	//Alarme Rosca de PO 1
	AL_RPO1 AT %QX3200.0:BOOL; 
	//Alarme Rosca de PO 2
	AL_RPO2 AT %QX3200.1:BOOL; 
	//Alarme Rosca de PO 3
	AL_RPO3 AT %QX3200.2:BOOL; 
	//Alarme Rosca de PO 4
	AL_RPO4 AT %QX3200.3:BOOL; 
	//Alarme Rosca de PO 5
	AL_RPO5 AT %QX3220.4:BOOL;
	//Alarme Rosca 6 Horizontal
	AL_RC6H AT %QX3200.5:BOOL; 
	//Alarme Rosca 7 Inclidada
	AL_RC7I AT %QX3200.6:BOOL;
	//Alarme Balança de solidos 1 descarga
	AL_BLS1D AT %QX3200.7:BOOL; 
	//Alarme Balança de solidos 2 descarga
	AL_BLS2D AT %QX3201.0:BOOL; 
	//Alarme Balança de solidos 3 descarga
	AL_BLS3D AT %QX3201.1:BOOL; 
	//Alarme Balança de solidos 4 descarga
	AL_BLS4D AT %QX3201.2:BOOL; 
	//Alarme Balança de solidos 5 descarga
	AL_BLS5D AT %QX3201.3:BOOL; 
	//Alarme Balança de liquidos 1 descarga
	AL_BL1D AT %QX3201.4:BOOL; 
	//Alarme Balança de liquidos 2 descarga
	AL_BL2D AT %QX3201.5:BOOL; 
	//Alarme Balança de liquidos 3 descarga
	AL_BL3D AT %QX3201.6:BOOL; 
	//Alarme Balança de liquidos 4 descarga
	AL_BL4D AT %QX3201.7:BOOL; 
	//Alarme Balança de liquidos 1 rapida
	AL_BLL1R AT %QX3202.0:BOOL; 
	//Alarme Balança de liquidos 1 lenta
	AL_BLL1L AT %QX3202.1:BOOL; 
	//Alarme Balança de liquidos 2 rapida ]
	AL_BLL2R AT %QX3202.2:BOOL;
	//Alarme Balança de liquidos 2 lenta
	AL_BLL2L AT %QX3202.3:BOOL;
	//Alarme Balança de liquidos 3 rapida
	AL_BLL3R AT %QX3202.4:BOOL; 
	//Alarme Balança de liquidos 3 lenta
	AL_BLL3L AT %QX3202.5:BOOL; 
	//Alarme Balança de liquidos 4 rapida
	AL_BLL4R AT %QX3202.6:BOOL; 
	//Alarme Balança de liquidos 4 lenta
	AL_BLL4L AT %QX3202.7:BOOL; 
	//Alarme Mexedor principal
	AL_CFMXP AT %QX3203.0:BOOL; 
	//Alarme Mexedor espera
	AL_MXE AT %QX3203.1:BOOL; 
	//Alarme Bomba oleo combuALivel
	AL_BOCOMB AT %QX3203.2:BOOL; 
	//Alarme Bomba diesel para piloto
	AL_BDP AT %QX3203.3:BOOL; 
	//Alarme Bomba de baixa ligada
	AL_BB AT %QX3203.4:BOOL;
	//Alarme Bomba de alta 1
	AL_BA1 AT %QX3203.5:BOOL; 
	//Alarme Bomba de alta 2
	AL_BA2 AT %QX3203.6:BOOL; 
	//Alarme Bomba de alta 3
	AL_BA3 AT %QX3203.7:BOOL; 
	//Alarme Moinho - Estrela
	AL_MHE AT %QX3204.0:BOOL; 
	//Alarme Exaustor estrela FM1
	AL_EXFM1_E AT %QX3204.1:BOOL; 
	//Alarme Exaustor FM2
	AL_EXFM2 AT %QX3204.2:BOOL; 
	//Alarme Exaustor FM3
	AL_EXFM3 AT %QX3204.3:BOOL; 
	//Alarme Esteira TC3 Dry Mix
	AL_TC3 AT %QX3204.4:BOOL; 
	//Alarme Esteira saida Air Lifit
	AL_ESTSAIRLF AT %QX3204.5:BOOL; 
	//Alarme Air Lifit
	AL_AIRLF AT %QX3204.6:BOOL;
	//Alarme Elevador 2
	AL_EL2 AT %QX3204.7:BOOL; 
	//Alarme Esteira TC8
	AL_ESTTC8 AT %QX3205.0:BOOL;
	//Alarme falta de pressão bomba de alta 1
	AL_FPBA1 AT %QX3205.1:BOOL;
	//Alarme falta de pressão bomba de alta 2
	AL_FPBA2 AT %QX3205.2:BOOL;
	//Alarme Moinho - Triangulo
	AL_MHT AT %QX3205.3:BOOL; 
	//Alarme valvula retorno não abriu
	AL_VLRNA AT %QX3205.4:BOOL;
	//Alarme valvula retorno não fechou
	AL_VLRNF AT %QX3205.5:BOOL;
	//Alarme bomba de transferencia
	AL_BBTRANS AT %QX3205.6:BOOL;
	//Alarme Exaustor triangulo FM1
	AL_EXFM1_T AT %QX3205.7:BOOL; 
	//Alarme bomba Blend	
	AL_BBLEND AT %QX3206.0:BOOL;
	//Alarme bomba Silicato
	AL_SILI AT %QX3206.1:BOOL;
	//Alarme exaustor da torre
	AL_EXTORRE AT %QX3206.2:BOOL;	
	//Alarme geral
	AL_GERAL AT %QX3206.3:BOOL;	
	//Alarme ventilador queimador
	AL_VENTQUEIMADOR AT %QX3206.4:BOOL;
	//Alarme falta oleo bomba alimentacao
	AL_BOCOMBFALT AT %QX3206.5:BOOL;
	//Alarme Exaustor estrela FM2
	AL_EXFM2_E AT %QX3206.6:BOOL; 		
	//Alarme Exaustor triangulo FM2
	AL_EXFM2_T AT %QX3206.7:BOOL;
	//Alarme Ventilador estrela FM2
	AL_VEXFM2_E AT %QX3207.0:BOOL; 		
	//Alarme Ventilador triangulo FM2
	AL_VEXFM2_T AT %QX3207.1:BOOL;
	//Alarme Peneira 1 não ligou
	AL_PN1 AT %QX3207.2:BOOL;	
	//Alarme Peneira 2 não ligou
	AL_PN2 AT %QX3207.3:BOOL;
	//Alarme Peneira 3 não ligou
	AL_PN3 AT %QX3207.4:BOOL;
	//Alarme Peneira 4 não ligou
	AL_PN4 AT %QX3207.5:BOOL;	
	//Alarme esteira saida torre não ligou
	AL_ESTSAITORRE AT %QX3207.6:BOOL;	
	//Alarme tempo de descarga balança de solido 1 ultrapassado
	AL_DESCARGA_BLS1 AT %QX3207.7:BOOL;		
	//Alarme tempo de descarga balança de solido 2 ultrapassado
	AL_DESCARGA_BLS2 AT %QX3208.0:BOOL;		
	//Alarme tempo de descarga balança de solido 3 ultrapassado
	AL_DESCARGA_BLS3 AT %QX3208.1:BOOL;		
	//Alarme tempo de descarga balança de solido 4 ultrapassado
	AL_DESCARGA_BLS4 AT %QX3208.2:BOOL;
	//Alarme tempo de descarga balança de solido 5 ultrapassado		
	AL_DESCARGA_BLS5 AT %QX3208.3:BOOL;
	//Alarme tempo de descarga balança de liquidos 1 ultrapassado		
	AL_DESCARGA_BLL1 AT %QX3208.4:BOOL;	
	//Alarme tempo de descarga balança de liquidos 2 ultrapassado	
	AL_DESCARGA_BLL2 AT %QX3208.5:BOOL;		
	//Alarme tempo de descarga balança de liquidos 3 ultrapassado
	AL_DESCARGA_BLL3 AT %QX3208.6:BOOL;		
	//Alarme tempo de descarga balança de liquidos 4 ultrapassado
	AL_DESCARGA_BLL4 AT %QX3208.7:BOOL;	
	//Alarme no sistema do queimador
	AL_QUEIMADOR AT %QX3209.0:BOOL;
	//Alarme Bomba de Sulfonico		
	AL_BBSULFONICO AT %QX3209.1:BOOL;
	//Alarme Bomba de Agua		
	AL_BBAGUA AT %QX3209.2:BOOL;
	//Alarme Bomba de Soda		
	AL_BBSODA AT %QX3209.3:BOOL;	
	//Alarme Peso alto BLS1
	AL_PESO_ALTO_BLS1 AT %QX3209.4:BOOL;		
	//Alarme Peso alto BLS2
	AL_PESO_ALTO_BLS2 AT %QX3209.5:BOOL;
	//Alarme Peso alto BLS3
	AL_PESO_ALTO_BLS3 AT %QX3209.6:BOOL;
	//Alarme Peso alto BLS4
	AL_PESO_ALTO_BLS4 AT %QX3209.7:BOOL;
	//Alarme Peso alto BLS5
	AL_PESO_ALTO_BLS5 AT %QX3210.0:BOOL;
	//Alarme Peso alto BLL1
	AL_PESO_ALTO_BLL1 AT %QX3210.1:BOOL;
	//Alarme Peso alto BLL2
	AL_PESO_ALTO_BLL2 AT %QX3210.2:BOOL;		
	//Alarme Peso alto BLL3
	AL_PESO_ALTO_BLL3 AT %QX3210.3:BOOL;			
	//Alarme Peso alto BLL4
	AL_PESO_ALTO_BLL4 AT %QX3210.4:BOOL;
	//Alarme Alta Temperatura Torre		
	AL_ALTA_TEMPE_TORRE AT %QX3210.5:BOOL;	
	//Y08 Comm.-Error Host  DS01 (Erro de Comunicação)	
	AL_SY08COMM_ERRORHOST_DS01 AT %QX3210.6:BOOL;
	//SY08 Comm.-Error Host  DS2 (Erro de Comunicação)	
	AL_SY08COMM_ERRORHOST_DS02 AT %QX3210.7:BOOL;		
	//SY08 Comm.-Error Host  DS3 (Erro de Comunicação)	
	AL_SY08COMM_ERRORHOST_DS03 AT %QX3211.0:BOOL;
	//SY08 Comm.-Error Host  DS4 (Erro de Comunicação)	
	AL_SY08COMM_ERRORHOST_DS04 AT %QX3211.1:BOOL;
	//SY08 Comm.-Error Host  DS5 (Erro de Comunicação)	
	AL_SY08COMM_ERRORHOST_DS05 AT %QX3211.2:BOOL;
	//SY08 Comm.-Error Host  DS7 (Erro de Comunicação)	
	AL_SY08COMM_ERRORHOST_DS07 AT %QX3211.3:BOOL;
	//SY08 Comm.-Error Host  DS8 (Erro de Comunicação)	
	AL_SY08COMM_ERRORHOST_DS08 AT %QX3211.4:BOOL;	
	//SY08 Comm.-Error Host  DS9 (Erro de Comunicação)	
	AL_SY08COMM_ERRORHOST_DS09 AT %QX3211.5:BOOL;		
	//SY08 Comm.-Error Host  DS10 (Erro de Comunicação)	
	AL_SY08COMM_ERRORHOST_DS10 AT %QX3211.6:BOOL;		
	//SY08 Comm.-Error Host  DS11 (Erro de Comunicação)	
	AL_SY08COMM_ERRORHOST_DS11 AT %QX3211.7:BOOL;	
	//SY08 Comm.-Error Host  DS12 (Erro de Comunicação)	
	AL_SY08COMM_ERRORHOST_DS12 AT %QX3212.0:BOOL;		
	//SY08 Comm.-Error Host  DS12 (Erro de Comunicação)	
	AL_SY08COMM_ERRORHOST_DS14 AT %QX3220.0:BOOL;		
	//SY08 Comm.-Error Host  DSTORRE (Erro de Comunicação)	
	AL_SY08COMM_ERRORHOST_DSTORRE AT %QX3212.1:BOOL;		
	//SC05 External Event1  DS01 (Falha acionamento Inversor)
	AL_SC05EXTERNAL_EVENT_DS01 AT %QX3212.2:BOOL;		
	//SC05 External Event1  DS2 (Falha acionamento Inversor)
	AL_SC05EXTERNAL_EVENT_DS02 AT %QX3212.3:BOOL;		
	//SC05 External Event1  DS3 (Falha acionamento Inversor)
	AL_SC05EXTERNAL_EVENT_DS03 AT %QX3212.4:BOOL;		
	//SC05 External Event1  DS4 (Falha acionamento Inversor)
	AL_SC05EXTERNAL_EVENT_DS04 AT %QX3212.5:BOOL;	
	//SC05 External Event1  DS5 (Falha acionamento Inversor)
	AL_SC05EXTERNAL_EVENT_DS05 AT %QX3212.6:BOOL;		
	//SC05 External Event1  DS7 (Falha acionamento Inversor)
	AL_SC05EXTERNAL_EVENT_DS07 AT %QX3212.7:BOOL;		
	//SC05 External Event1  DS8 (Falha acionamento Inversor)
	AL_SC05EXTERNAL_EVENT_DS08 AT %QX3213.0:BOOL;		
	//SC05 External Event1  DS9 (Falha acionamento Inversor)
	AL_SC05EXTERNAL_EVENT_DS09 AT %QX3213.1:BOOL;		
	//SC05 External Event1  DS10 (Falha acionamento Inversor)
	AL_SC05EXTERNAL_EVENT_DS10 AT %QX3213.2:BOOL;		
	//SC05 External Event1  DS11 (Falha acionamento Inversor)
	AL_SC05EXTERNAL_EVENT_DS11 AT %QX3213.3:BOOL;		
	//SC05 External Event1  DS12 (Falha acionamento Inversor)
	AL_SC05EXTERNAL_EVENT_DS12 AT %QX3213.4:BOOL;		
	//SC05 External Event1  DS12 (Falha acionamento Inversor)
	AL_SC05EXTERNAL_EVENT_DS14 AT %QX3220.1:BOOL;		
	//SC05 External Event1  DTORRE (Falha acionamento Inversor)
	AL_SC05EXTERNAL_EVENT_DSTORRE AT %QX3213.5:BOOL;		
	//SC09 Feedback Gate  DS01 (Confirmação Valvula Fechada)
	AL_SC09FEEDDBACK_GATE_DS01 AT %QX3213.6:BOOL;		
	//SC09 Feedback Gate  DS2 (Confirmação Valvula Fechada)
	AL_SC09FEEDDBACK_GATE_DS02 AT %QX3213.7:BOOL;	
	//SC09 Feedback Gate  DS3 (Confirmação Valvula Fechada)
	AL_SC09FEEDDBACK_GATE_DS03 AT %QX3214.0:BOOL;		
	//SC09 Feedback Gate  DS4 (Confirmação Valvula Fechada)	 
	AL_SC09FEEDDBACK_GATE_DS04 AT %QX3214.1:BOOL;	
	//SC09 Feedback Gate  DS5 (Confirmação Valvula Fechada)
	AL_SC09FEEDDBACK_GATE_DS05 AT %QX3214.2:BOOL;		
	//SC09 Feedback Gate DS7 (Confirmação Valvula Fechada)
	AL_SC09FEEDDBACK_GATE_DS07 AT %QX3214.3:BOOL;	  	
	//SC09 Feedback Gate  DS8 (Confirmação Valvula Fechada)
	AL_SC09FEEDDBACK_GATE_DS08 AT %QX3214.4:BOOL;		
	//SC09 Feedback Gate  DS9 (Confirmação Valvula Fechada)
	AL_SC09FEEDDBACK_GATE_DS09 AT %QX3214.5:BOOL;		
	//SC09 Feedback Gate  DS10 (Confirmação Valvula Fechada)
	AL_SC09FEEDDBACK_GATE_DS10 AT %QX3214.6:BOOL;		
	//SC09 Feedback Gate  Ds11 (Confirmação Valvula Fechada)
	AL_SC09FEEDDBACK_GATE_DS11 AT %QX3214.7:BOOL;		
	//SC09 Feedback Gate  DS12 (Confirmação Valvula Fechada)
	AL_SC09FEEDDBACK_GATE_DS12 AT %QX3215.0:BOOL;		
	//SC09 Feedback Gate  DS12 (Confirmação Valvula Fechada)
	AL_SC09FEEDDBACK_GATE_DS14 AT %QX3220.2:BOOL;		
	//SC09 Feedback Gate  DSTORRE (Confirmação Valvula Fechada)
	AL_SC09FEEDDBACK_GATE_DSTORRE AT %QX3215.1:BOOL;		
	//HI05 Control Deviation DS01 (Controle de Desvio)
	AL_HI05_CONTROL_DEVIATION_DS01 AT %QX3215.2:BOOL;		
	//HI05 Control Deviation DS02 (Controle de Desvio)
	AL_HI05_CONTROL_DEVIATION_DS02 AT %QX3215.3:BOOL;		
	//HI05 Control Deviation DS03 (Controle de Desvio)
	AL_HI05_CONTROL_DEVIATION_DS03 AT %QX3215.4:BOOL;		
	//HI05 Control Deviation DS04 (Controle de Desvio)
	AL_HI05_CONTROL_DEVIATION_DS04 AT %QX3215.5:BOOL;		
	//HI05 Control Deviation DS05 (Controle de Desvio)
	AL_HI05_CONTROL_DEVIATION_DS05 AT %QX3215.6:BOOL;	
	//HI05 Control Deviation DS07 (Controle de Desvio)
	AL_HI05_CONTROL_DEVIATION_DS07 AT %QX3215.7:BOOL;	
	//HI05 Control Deviation DS08 (Controle de Desvio)
	AL_HI05_CONTROL_DEVIATION_DS08 AT %QX3216.0:BOOL;		
	//HI05 Control Deviation DS09 (Controle de Desvio)
	AL_HI05_CONTROL_DEVIATION_DS09 AT %QX3216.1:BOOL;		
	//HI05 Control Deviation DS10 (Controle de Desvio)
	AL_HI05_CONTROL_DEVIATION_DS10 AT %QX3216.2:BOOL;	
	//HI05 Control Deviation DS11 (Controle de Desvio)
	AL_HI05_CONTROL_DEVIATION_DS11 AT %QX3216.3:BOOL;		
	//HI05 Control Deviation DS12 (Controle de Desvio)
	AL_HI05_CONTROL_DEVIATION_DS12 AT %QX3216.4:BOOL;		
	// HI05 Control Deviation DS14 (Controle de Desvio)
	AL_HI05_CONTROL_DEVIATION_DS14 AT %QX3220.3:BOOL;		
	//HI05 Control Deviation DSTORRE (Controle de Desvio)
	AL_HI05_CONTROL_DEVIATION_DSTORRE AT %QX3216.5:BOOL;		
	


	//WORD - bloco 1 de alarmes
	Alarmes1 AT %QW3150:WORD;
	//WORD - bloco 2 de alarmes
	Alarmes2 AT %QW3152:WORD;
	//WORD - bloco 3 de alarmes
	Alarmes3 AT %QW3154:WORD;
	//WORD - bloco 4 de alarmes
	Alarmes4 AT %QW3156:WORD;
	//WORD - bloco 5 de alarmes
	Alarmes5 AT %QW3158:WORD;
	//WORD - bloco 6 de alarmes
	Alarmes6 AT %QW3160:WORD;
	//WORD - bloco 7 de alarmes
	Alarmes7 AT %QW3162:WORD;
	//WORD - bloco 8 de alarmes
	Alarmes8 AT %QW3164:WORD;
	//WORD - bloco 9 de alarmes
	Alarmes9 AT %QW3166:WORD;

	//Silencia alarme alta temperatura da torre
	SILENCIA_AL_ALTA_TEMPE_TORRE:BOOL;

	
END_VAR

// Device/Application/GVLGerais
//Global Variable List de comando do supervisório
VAR_GLOBAL
	
	//Botão liga Bomba oleo combustivel	 
	BTS_BOCOMB	AT	%QX3003.2	:BOOL;
	//Botão liga Bomba diesel para piloto	 
	BTS_BDP	AT	%QX3003.3	:BOOL;
	// Botão reset alarmes
	BTS_RSTAL AT %QX3005.0 :BOOL;
	
	BTS_RESERVA1 AT	%QX3020.2:BOOL;
	BTS_RESERVA2 AT	%QX3020.3:BOOL;
	BTS_RESERVA3 AT	%QX3020.4:BOOL;
	BTS_RESERVA4 AT	%QX3020.5:BOOL;
	BTS_RESERVA5 AT	%QX3020.6:BOOL;
	BTS_RESERVA6 AT	%QX3020.7:BOOL;
	BTS_BB_AUTOM AT	%QX3021.0:BOOL;
	BB_AUTOM AT	%QX3021.1:BOOL;
	BTS_RESERVA9 AT	%QX3021.2:BOOL;
	BTS_RESERVA10 AT %QX3021.3:BOOL;
	BTS_RESERVA11 AT %QX3021.4:BOOL;
	BTS_RESERVA12 AT %QX3021.5:BOOL;
	BTS_RESERVA13 AT %QX3021.6:BOOL;
	BTS_RESERVA14 AT %QX3021.7:BOOL;
	BTS_RESERVA15 AT %QX3022.0:BOOL;
	BTS_RESERVA16 AT %QX3022.1:BOOL;
	BTS_RESERVA17 AT %QX3022.2:BOOL;
	BTS_RESERVA18 AT %QX3022.3:BOOL;
	BTS_RESERVA19 AT %QX3022.4:BOOL;
	BTS_RESERVA20 AT %QX3022.5:BOOL;
	BTS_RESERVA21 AT %QX3022.6:BOOL;
	BTS_RESERVA22 AT %QX3022.7:BOOL;
	BTS_RESERVA23 AT %QX3023.0:BOOL;
	BTS_RESERVA24 AT %QX3023.1:BOOL;
	BTS_RESERVA25 AT %QX3023.2:BOOL;
	BTS_RESERVA26 AT %QX3023.3:BOOL;
	BTS_RESERVA27 AT %QX3023.4:BOOL;
	BTS_RESERVA28 AT %QX3023.5:BOOL;
	BTS_RESERVA29 AT %QX3023.6:BOOL;
	BTS_RESERVA30 AT %QX3023.7:BOOL;
	BTS_RESERVA31 AT %QX3024.0:BOOL;
	BTS_RESERVA32 AT %QX3024.1:BOOL;
	BTS_RESERVA33 AT %QX3024.2:BOOL;
	BTS_RESERVA34 AT %QX3024.3:BOOL;
	BTS_RESERVA35 AT %QX3024.4:BOOL;
	BTS_RESERVA36 AT %QX3024.5:BOOL;
	BTS_RESERVA37 AT %QX3024.6:BOOL;
	BTS_RESERVA38 AT %QX3024.7:BOOL;
	
	//======VARIÁVEIS DE COMUNICAÇÃO COM SUPERVISÓRIO PARA CÁLCULO DE OEE
	
	
	//======VARIÁVEIS DE COMUNICAÇÃO L1
	//Contador de produção L1
	CNT_PRD_L1_1T AT %QD10240: INT;
	//Eficiência PROJETADA para linha 1 até o momento atual.
	EficL1_1T_projetada AT %QD10280: REAL;
	//Eficiência REAL para linha 1 até o momento atual.
	EficL1_1T_realtime AT %QD10588: REAL;
	//Produção programada pelo PCP no 1º turno
	ProducaoProgramada_L1_1T AT %QD10360: INT;
	//Produção programada pelo PCP no 2º turno
	ProducaoProgramada_L1_2T  AT %QD10484: INT;
	//Produção programada pelo PCP no 3º turno
	ProducaoProgramada_L1_3T  AT %QD10524: INT;
	TempoParada AT %QD10592: INT;
	TempoProduzindo AT %QD10480: INT;
	CXS_ATRASOL1 AT %QD10696: INT;
	//======VARIÁVEIS DE COMUNICAÇÃO L2
	
	//======VARIÁVEIS DE COMUNICAÇÃO L2
	//Contador de produção L2
	CNT_PRD_L2_1T AT %QD10244: INT;
	//Eficiência PROJETADA para linha 2 até o momento atual.
	EficL2_1T_projetada AT %QD10284: REAL;
	//Eficiência REAL para linha 2 até o momento atual.
	EficL2_1T_realtime AT %QD10420: REAL;
	//Produção programada pelo PCP no 1º turno
	ProducaoProgramada_L2_1T AT %QD10364: INT;
	//Produção programada pelo PCP no 2º turno
	ProducaoProgramada_L2_2T  AT %QD10488: INT;
	//Produção programada pelo PCP no 3º turno
	ProducaoProgramada_L2_3T  AT %QD10524: INT;
	TempoParadaL2 AT %QD10596: INT;
	TempoProduzindoL2 AT %QD10600: INT;
	CXS_ATRASOL2 AT %QD10700: INT;
	//======VARIÁVEIS DE COMUNICAÇÃO L2
	
		//======VARIÁVEIS DE COMUNICAÇÃO L3
	//Contador de produção L1
	CNT_PRD_L3_1T AT %QD10248: INT;
	//Eficiência PROJETADA para linha 1 até o momento atual.
	EficL3_1T_projetada AT %QD10288: REAL;
	//Eficiência REAL para linha 1 até o momento atual.
	EficL3_1T_realtime AT %QD10424: REAL;
	//Produção programada pelo PCP no 1º turno
	ProducaoProgramada_L3_1T AT %QD10368: INT;
	//Produção programada pelo PCP no 2º turno
	ProducaoProgramada_L3_T2 AT %QD10492: INT;
	//Produção programada pelo PCP no 3º turno
	ProducaoProgramada_L3_T3 AT %QD10532: INT;
	TempoParadaL3 AT %QD10640: INT;
	TempoProduzindoL3 AT %QD10644: INT;
	CXS_ATRASOL3 AT %QD10704: INT;

	//======VARIÁVEIS DE COMUNICAÇÃO L3
	
		//======VARIÁVEIS DE COMUNICAÇÃO L4
	//Contador de produção L1
	CNT_PRD_L4_1T AT %QD10252: INT;
	//Eficiência PROJETADA para linha 1 até o momento atual.
	EficL4_1T_projetada AT %QD10292: REAL;
	//Eficiência REAL para linha 1 até o momento atual.
	EficL4_1T_realtime AT %QD10428: REAL;
	//Produção programada pelo PCP no 1º turno
	ProducaoProgramada_L4_1T AT %QD10372: INT;
	//Produção programada pelo PCP no 2º turno
	ProducaoProgramada_L4_T2 AT %QD10496: INT;
	//Produção programada pelo PCP no 3º turno
	ProducaoProgramada_L4_T3 AT %QD10536: INT;
	TempoParadaL4 AT %QD10648: INT;
	TempoProduzindoL4 AT %QD10652: INT;
	CXS_ATRASOL4 AT %QD10708: INT;

	//======VARIÁVEIS DE COMUNICAÇÃO L4
	
		//======VARIÁVEIS DE COMUNICAÇÃO L5
	//Contador de produção L1
	CNT_PRD_L5_1T AT %QD10256: INT;
	//Eficiência PROJETADA para linha 1 até o momento atual.
	EficL5_1T_projetada AT %QD10296: REAL;
	//Eficiência REAL para linha 1 até o momento atual.
	EficL5_1T_realtime AT %QD10432: REAL;
	//Produção programada pelo PCP no 1º turno
	ProducaoProgramada_L5_1T AT %QD10376: INT;
	//Produção programada pelo PCP no 1º turno
	ProducaoProgramada_L5_T2 AT %QD10500: INT;
	//Produção programada pelo PCP no 1º turno
	ProducaoProgramada_L5_T3 AT %QD10540: INT;
	TempoParadaL5 AT %QD10656: INT;
	TempoProduzindoL5 AT %QD10660: INT;
	CXS_ATRASOL5 AT %QD10712: INT;
	
	//======VARIÁVEIS DE COMUNICAÇÃO L5
	
	//======VARIÁVEIS DE COMUNICAÇÃO L6
	//Contador de produção L6
	CNT_PRD_L6_1T AT %QD10260: INT;
	//Eficiência PROJETADA para linha 1 até o momento atual.
	EficL6_1T_projetada AT %QD10400: REAL;
	//Eficiência REAL para linha 1 até o momento atual.
	EficL6_1T_realtime AT %QD10436: REAL;
	//Produção programada pelo PCP no 1º turno
	ProducaoProgramada_L6_1T AT %QD10464: INT;
	//Produção programada pelo PCP no 1º turno
	ProducaoProgramada_L6_T2 AT %QD10504: INT;
	//Produção programada pelo PCP no 1º turno
	ProducaoProgramada_L6_T3 AT %QD10544: INT;
	TempoParadaL6 AT %QD10664: INT;
	TempoProduzindoL6 AT %QD10668: INT;
	CXS_ATRASOL6 AT %QD10716: INT;
	//======VARIÁVEIS DE COMUNICAÇÃO L6
	
		//======VARIÁVEIS DE COMUNICAÇÃO L7
	//Contador de produção L7
	CNT_PRD_L7_1T AT %QD10264: INT;
	//Eficiência PROJETADA para linha 1 até o momento atual.
	EficL7_1T_projetada AT %QD10404: REAL;
	//Eficiência REAL para linha 1 até o momento atual.
	EficL7_1T_realtime AT %QD10440: REAL;
	//Produção programada pelo PCP no 1º turno
	ProducaoProgramada_L7_1T AT %QD10468: INT;
	//Produção programada pelo PCP no 1º turno
	ProducaoProgramada_L7_T2 AT %QD10508: INT;
	//Produção programada pelo PCP no 1º turno
	ProducaoProgramada_L7_T3 AT %QD10624: INT;
	TempoParadaL7 AT %QD10672: INT;
	TempoProduzindoL7 AT %QD10676: INT;
	CXS_ATRASOL7 AT %QD10720: INT;
	//======VARIÁVEIS DE COMUNICAÇÃO L7
	
		//======VARIÁVEIS DE COMUNICAÇÃO L8
	//Contador de produção L8
	CNT_PRD_L8_1T AT %QD10268: INT;
	//Eficiência PROJETADA para linha 1 até o momento atual.
	EficL8_1T_projetada AT %QD10408: REAL;
	//Eficiência REAL para linha 1 até o momento atual.
	EficL8_1T_realtime AT %QD10348: REAL;
	//Produção programada pelo PCP no 1º turno
	ProducaoProgramada_L8_1T AT %QD10472: INT;
	//Produção programada pelo PCP no 1º turno
	ProducaoProgramada_L8_T2 AT %QD10512: INT;
	//Produção programada pelo PCP no 1º turno
	ProducaoProgramada_L8_T3 AT %QD10552: INT;
	TempoParadaL8 AT %QD10680: INT;
	TempoProduzindoL8 AT %QD10684: INT;
	CXS_ATRASOL8 AT %QD10724: INT;
	//======VARIÁVEIS DE COMUNICAÇÃO L8
	
		//======VARIÁVEIS DE COMUNICAÇÃO L9
	//Contador de produção L9
	CNT_PRD_L9_1T AT %QD10272: INT;
	//Eficiência PROJETADA para linha 1 até o momento atual.
	EficL9_1T_projetada AT %QD10412: REAL;
	//Eficiência REAL para linha 1 até o momento atual.
	EficL9_1T_realtime AT %QD10352: REAL;
	//Produção programada pelo PCP no 1º turno
	ProducaoProgramada_L9_1T AT %QD10476: INT;
	//Produção programada pelo PCP no 1º turno
	ProducaoProgramada_L9_T2 AT %QD10516: INT;
	//Produção programada pelo PCP no 1º turno
	ProducaoProgramada_L9_T3 AT %QD10556: INT;
	TempoParadaL9 AT %QD10688: INT;
	TempoProduzindoL9 AT %QD10692: INT;
	CXS_ATRASOL9 AT %QD10728: INT;
	//======VARIÁVEIS DE COMUNICAÇÃO L9
	
	//======HORÁRIOS E STATUS DE PRODUÇÃO
	HoraInicio1Turno AT %QD10356  : INT;
MinInicio1Turno AT %QD10568 : INT;
HoraInicio2Turno AT %QD10572 :  INT;
MinInicio2Turno AT %QD10576 :  INT;
HoraInicio3Turno AT %QD10580 : INT;
MinInicio3Turno AT%QD10584 : INT;
MinDispTurnoAtual AT %QD10276 : REAL;
Status_L1 AT %QD10416: INT;
Status_L2 AT %QD10604: INT;
Status_L3 AT %QD10608: INT;
Status_L4 AT %QD10612: INT;
Status_L5 AT %QD10616: INT;
Status_L6 AT %QD10620: INT;
Status_L7 AT %QD10624: INT;
Status_L8 AT %QD10628: INT;
Status_L9 AT %QD10632: INT;
StatusLAerossol AT %QD10636: INT;



//======HORÁRIO DE INICIO E FIM DE CADA TURNO	
	
END_VAR

// Device/Application/GVLSlurryMaking
VAR_GLOBAL
	// boleanos
	
	//Botão liga  Rosca de PO 1
	BTS_RPO1	AT	%QX3000.0	:BOOL;
	//Botão liga  Rosca de PO 2	 
	BTS_RPO2	AT	%QX3000.1	:BOOL;
	//Botão liga  Rosca de PO 3 	 
	BTS_RPO3	AT	%QX3000.2	:BOOL;	
	//Botão liga Rosca de PO 4
	BTS_RPO4	AT	%QX3000.3	:BOOL;
	//Botão liga Rosca de PO 5	 
	BTS_RPO5	AT	%QX3000.4	:BOOL;	
	//Botão liga Rosca 6 Horizontal 
	BTS_RC6H	AT	%QX3000.5	:BOOL;
	//Botão liga Rosca 7 Inclidada	
	BTS_RC7I	AT	%QX3000.6	:BOOL;	
	//Botão liga  Balança de solidos 1 descarga 
	BTS_BLS1D	AT	%QX3000.7	:BOOL;	
	//Botão liga Balança de solidos 2 descarga
	BTS_BLS2D	AT	%QX3001.0	:BOOL;	
	//Botão liga Balança de solidos 3 descarga  
	BTS_BLS3D	AT	%QX3001.1	:BOOL;	
	//Botão liga Balança de solidos 4 descarga 
	BTS_BLS4D	AT	%QX3001.2	:BOOL;
	//Botão liga Balança de solidos 5 descarga	
	BTS_BLS5D	AT	%QX3001.3	:BOOL;	
	//Botão liga Balança de liquidos 1 descarga 
	BTS_BL1D	AT	%QX3001.4	:BOOL;	
	//Botão liga Balança de liquidos 2 descarga  
	BTS_BL2D	AT	%QX3001.5	:BOOL;
	//Botão liga Balança de liquidos 3 descarga 	
	BTS_BL3D	AT	%QX3001.6	:BOOL;
	//Botão liga Balança de liquidos 4 descarga	
	BTS_BL4D	AT	%QX3001.7	:BOOL;	
	//Botão liga Balança de liquidos 1 rapida 
	BTS_BLL1R	AT	%QX3002.0	:BOOL;
	//Botão liga Balança de liquidos 1 lenta 	 
	BTS_BLL1L	AT	%QX3002.1	:BOOL;
	//Botão liga Balança de liquidos 2 rapida 	
	BTS_BLL2R	AT	%QX3002.2	:BOOL;
	//Botão liga Balança de liquidos 2 lenta 	
	BTS_BLL2L	AT	%QX3002.3	:BOOL;
	//Botão liga Balança de liquidos 3 rapida 	
	BTS_BLL3R 	AT	%QX3002.4	:BOOL;
	//Botão liga Balança de liquidos 3 lenta	
	BTS_BLL3L	AT	%QX3002.5	:BOOL;
	//Botão liga Balança de liquidos 4 rapida	 
	BTS_BLL4R	AT	%QX3002.6	:BOOL;
	//Botão liga Balança de liquidos 4 lenta	 
	BTS_BLL4L 	AT	%QX3002.7	:BOOL;
	//Botão liga Mexedor principal	 
	BTS_CFMXP	AT	%QX3003.0	:BOOL;
	//SET PARA REGISTRA HISTORICO DE PESO DO MISTURADOR
	VAL_REG_PESO_MSP AT %QX3009.6: BOOL;
	//Botão zera posição equipamento
	BTS_ZERAPS AT %QX3005.5:BOOL;	
	//Botão manual/automatico off/on Slurry Making
	BTS_MASLU AT %QX3005.6:BOOL;	
	//Botão liga aquecimento no mexedor principal
	BTS_AQUEMXP AT %QX3006.0:BOOL;
	//Botão liga bomba de agua
	BTS_BAG AT %QX3006.1:BOOL;
	//Botão liga valvula de saida do misturador principal
	BTS_VLSMXP AT %QX3006.2:BOOL;	
	//Botão zera fluximetro agua
	BTS_ZERAFLUXIMETRO AT %QX3017.4:BOOL;	
	//Botão inicio ciclo
	BTS_INICICLO AT %QX3005.3:BOOL;		
	//Botão parada de ciclo
	BTS_PARADA_CICLO AT	%QX3017.5:BOOL;	
	//Botão ultima carga Slurry
	BTS_ULTIMA_CARGA AT %QX3017.6:BOOL;			
	//Botão liga Botão liga Bomba Acusol	 
	BTS_BACU AT	%QX3003.7	:BOOL;
	//Transferencia liberada
	TRANSFERENCIA_lIBERADA:BOOL;
	//Ultima carga
	ULTIMA_CARGA:BOOL;
	//Botão Permite Descarga com peso Maximo BLS1
	BTS_PERMI_DESCAR_PESO_MAX_BLS1 AT %QX3018.7:BOOL;		
	//Botão Permite Descarga com peso Maximo BLS2
	BTS_PERMI_DESCAR_PESO_MAX_BLS2 AT %QX3019.0:BOOL;		
	//Botão Permite Descarga com peso Maximo BLS3
	BTS_PERMI_DESCAR_PESO_MAX_BLS3 AT %QX3019.1:BOOL;		
	//Botão Permite Descarga com peso Maximo BLS4
	BTS_PERMI_DESCAR_PESO_MAX_BLS4 AT %QX3019.2:BOOL;		
	//Botão Permite Descarga com peso Maximo BLS5
	BTS_PERMI_DESCAR_PESO_MAX_BLS5 AT %QX3019.3:BOOL;		
	//Botão Permite Descarga com peso Maximo BLL1
	BTS_PERMI_DESCAR_PESO_MAX_BLL1 AT %QX3019.4:BOOL;		
	//Botão Permite Descarga com peso Maximo BLL2
	BTS_PERMI_DESCAR_PESO_MAX_BLL2 AT %QX3019.5:BOOL;		
	//Botão Permite Descarga com peso Maximo BLL3
	BTS_PERMI_DESCAR_PESO_MAX_BLL3 AT %QX3019.6:BOOL;		
	//Botão Permite Descarga com peso Maximo BLL4
	BTS_PERMI_DESCAR_PESO_MAX_BLL4 AT %QX3019.7:BOOL;		
	// BLS1 CARREGADA
	BLS1_CARREGADA:BOOL;
	// BLS2 CARREGADA
	BLS2_CARREGADA:BOOL;
	// BLS3 CARREGADA
	BLS3_CARREGADA:BOOL;
	// BLS4 CARREGADA
	BLS4_CARREGADA:BOOL;
	// BLS5 CARREGADA
	BLS5_CARREGADA:BOOL;
	// BLL1 CARREGADA
	BLL1_CARREGADA:BOOL;
	// BLl2 CARREGADA
	BLL2_CARREGADA:BOOL;
	// BLl3 CARREGADA
	BLL3_CARREGADA:BOOL;
	// BLl4 CARREGADA
	BLL4_CARREGADA:BOOL;
	

	// registradores
	
	//Leitura Peso balança de solido 1
	LEITURA_PESO_BLS1 AT %QD13032:REAL;
	//Leitura Peso balança de solido 2
	LEITURA_PESO_BLS2 AT %QD13036:REAL;
	//Leitura Peso balança de solido 3
	LEITURA_PESO_BLS3 AT %QD13040:REAL;
	//Leitura Peso balança de solido 4
	LEITURA_PESO_BLS4 AT %QD13044:REAL;
	//Leitura Peso balança de solido 5
	LEITURA_PESO_BLS5 AT %QD13048:REAL;
	//Leitura Peso balança de liquido 1
	LEITURA_PESO_BLL1 AT %QD13052:REAL;
	//Leitura Peso balança de liquido 2
	LEITURA_PESO_BLL2 AT %QD13056:REAL;
	//Leitura Peso balança de liquido 3
	LEITURA_PESO_BLL3 AT %QD13060:REAL;
	//Leitura Peso balança de liquido 4
	LEITURA_PESO_BLL4 AT %QD13064:REAL;
	//Nivel Misturador Principal
	LEITURA_NI_MISTPRIN AT %QD13076:REAL;	
	//Quantidade de agua dosada
	QTD_AGUA_DOSADA AT %QD13120:REAL;
	//Programa carregado Slurry
	PROGRAMA_CARREGADO_SLURRY AT %QD12830:REAL;	
		
	//Leitura REAL engenharia BLS1
	LEITURA_REAL_ENGE_BLS1 AT %QD13152:REAL;		
	//Leitura REAL engenharia BLS2
	LEITURA_REAL_ENGE_BLS2 AT %QD13156:REAL;		
	//Leitura REAL engenharia BLS3
	LEITURA_REAL_ENGE_BLS3 AT %QD13160:REAL;		
	//Leitura REAL engenharia BLS4
	LEITURA_REAL_ENGE_BLS4 AT %QD13164:REAL;		
	//Leitura REAL engenharia BLS5
	LEITURA_REAL_ENGE_BLS5 AT %QD13168:REAL;		
	//Leitura REAL engenharia BLL1
	LEITURA_REAL_ENGE_BLL1 AT %QD13172:REAL;		
	//Leitura REAL engenharia BLL2
	LEITURA_REAL_ENGE_BLL2 AT %QD13176:REAL;		
	//Leitura REAL engenharia BLL3
	LEITURA_REAL_ENGE_BLL3 AT %QD13180:REAL;		
	//Leitura REAL engenharia BLL4
	LEITURA_REAL_ENGE_BLL4 AT %QD13184:REAL;	
	//Pesos gravado DO Slurry	
	LEITURA_STATUS_PESOS_SLURRY_GRAVADO AT %QD13244:REAL;
	//Preset Reset Status Leitura Pesos Slurry			
	PRST_RESET_STATUS_LEITURA_SLURRY AT %QD13556:REAL;	
	
	
END_VAR

VAR_GLOBAL PERSISTENT
	//Leitura sequencia atual
	LEITURA_SEQ_ATUAL AT %QD13148:REAL;	
	//Preset peso balança de solido 1
	PRST_PESO_BLS1 AT %QD12290:REAL;
	//Preset peso balança de solido 2
	PRST_PESO_BLS2 AT %QD12294:REAL;
	//Preset peso balança de solido 3
	PRST_PESO_BLS3 AT %QD12298:REAL;
	//Preset peso balança de solido 4
	PRST_PESO_BLS4 AT %QD12302:REAL;
	//Preset peso balança de solido 5
	PRST_PESO_BLS5 AT %QD12306:REAL;
	//Preset peso balança de liquido 1
	PRST_PESO_BLL1 AT %QD12310:REAL;
	//Preset peso balança de liquido 2
	PRST_PESO_BLL2 AT %QD12314:REAL;
	//Preset peso balança de liquido 3
	PRST_PESO_BLL3 AT %QD12318:REAL;
	//Preset peso balança de liquido 4
	PRST_PESO_BLL4 AT %QD12322:REAL;
	//Preset Peso Acusol, somando com peso do blend
	//PRST_PESO_ACUSOL AT %QD12574:REAL;		
	PRST_PESO_ACUSOL :REAL;
	
	//Zero Pesagem balanca solidos 1
	PRST_ZERO_PESO_BLS1 AT %QD12490:REAL;
	//Zero Pesagem balanca solidos 2		
	PRST_ZERO_PESO_BLS2 AT %QD12494:REAL;
	//Zero Pesagem balanca solidos 3		
	PRST_ZERO_PESO_BLS3 AT %QD12498:REAL;
	//Zero Pesagem balanca solidos 4		
	PRST_ZERO_PESO_BLS4 AT %QD12502:REAL;
	//Zero Pesagem balanca solidos 5		
	PRST_ZERO_PESO_BLS5 AT %QD12506:REAL;	
	//Zero Pesagem balanca liquidos 1	
	PRST_ZERO_PESO_BLL1 AT %QD12510:REAL;
	//Zero Pesagem balanca liquidos 2		
	PRST_ZERO_PESO_BLL2 AT %QD12514:REAL;
	//Zero Pesagem balanca liquidos 3		
	PRST_ZERO_PESO_BLL3 AT %QD12518:REAL;
	//Zero Pesagem balanca liquidos 4		
	PRST_ZERO_PESO_BLL4 AT %QD12522:REAL;		
	
	//Minimo peso balança de solido 1
	PRST_MIN_PESO_BLS1 AT %QD12326:REAL;
	//Minimo peso balança de solido 2
	PRST_MIN_PESO_BLS2 AT %QD12340:REAL;
	//Minimo peso balança de solido 3
	PRST_MIN_PESO_BLS3 AT %QD12344:REAL;
	//Minimo peso balança de solido 4
	PRST_MIN_PESO_BLS4 AT %QD12348:REAL;
	//Minimo peso balança de solido 5
	PRST_MIN_PESO_BLS5 AT %QD12352:REAL;
	//Minimo peso balança de liquido 1
	PRST_MIN_PESO_BLL1 AT %QD12356:REAL;
	//Minimo peso balança de liquido 2
	PRST_MIN_PESO_BLL2 AT %QD12360:REAL;
	//Minimo peso balança de liquido 3
	PRST_MIN_PESO_BLL3 AT %QD12364:REAL;
	//Minimo peso balança de liquido 4
	PRST_MIN_PESO_BLL4 AT %QD12368:REAL;
			
	//Porcentagem de erro Maximo peso balança de solido 1
	PRST_PORCENTAGEM_ERRO_PESO_BLS1 AT %QD12372:REAL;
	//Porcentagem de erro Maximo peso balança de solido 2
	PRST_PORCENTAGEM_ERRO_PESO_BLS2 AT %QD12376:REAL;
	//Porcentagem de erro Maximo peso balança de solido 3
	PRST_PORCENTAGEM_ERRO_PESO_BLS3 AT %QD12380:REAL;
	//Porcentagem de erro Maximo peso balança de solido 4
	PRST_PORCENTAGEM_ERRO_PESO_BLS4 AT %QD12384:REAL;
	//Porcentagem de erro Maximo peso balança de solido 5
	PRST_PORCENTAGEM_ERRO_PESO_BLS5 AT %QD12388:REAL;
	//Porcentagem de erro Maximo peso balança de liquido 1
	PRST_PORCENTAGEM_ERRO_PESO_BLL1 AT %QD12392:REAL;
	//Porcentagem de erro Maximo peso balança de liquido 2
	PRST_PORCENTAGEM_ERRO_PESO_BLL2 AT %QD12396:REAL;
	//Porcentagem de erro Maximo peso balança de liquido 3
	PRST_PORCENTAGEM_ERRO_PESO_BLL3 AT %QD12400:REAL;
	//Porcentagem de erro Maximo peso balança de liquido 4
	PRST_PORCENTAGEM_ERRO_PESO_BLL4 AT %QD12404:REAL;	
	//Quantidade de agua no MXP litros
	PRST_QNTDE_AGUA AT %QD12448:REAL;
	
	//Preset valor posicao sequencia Balança Solido 1
	PRST_POSSEQ_BLS1 AT %QW12460:INT;	
	//Preset valor posicao sequencia Balança Solido 2	
	PRST_POSSEQ_BLS2 AT %QW12462:INT;	
	//Preset valor posicao sequencia Balança Solido 3	
	PRST_POSSEQ_BLS3 AT %QW12464:INT;
	//Preset valor posicao sequencia Balança Solido 4		
	PRST_POSSEQ_BLS4 AT %QW12466:INT;		
	//Preset valor posicao sequencia Balança Solido 5
	PRST_POSSEQ_BLS5 AT %QW12468:INT;
	//Preset valor posicao sequencia Balança Liquidos 1		
	PRST_POSSEQ_BLL1 AT %QW12470:INT;	
	//Preset valor posicao sequencia Balança Liquidos 2	
	PRST_POSSEQ_BLL2 AT %QW12472:INT;		
	//Preset valor posicao sequencia Balança Liquidos 3
	PRST_POSSEQ_BLL3 AT %QW12474:INT;
	//Preset valor posicao sequencia Balança Liquidos 4		
	PRST_POSSEQ_BLL4 AT %QW12476:INT;
	//Preset valor posicao sequencia agua		
	PRST_POSSEQ_AGUA AT %QW12478:INT;
	//Preset valor posicao sequencia vapor		
	PRST_POSSEQ_VAPOR AT %QW12480:INT;		
	//Preset valor posicao sequencia saida misturador
	PRST_POSSEQ_VALSAIDA_MXP AT %QW12482:INT;
	//Preset valor posicao sequencia tempo reação		
	PRST_POSSEQ_TEMPO_REACAO AT %QW12484:INT;		
	//Preset valor posicao sequencia tempo hidratação
	PRST_POSSEQ_TEMPO_HIDRATA AT %QW12486:INT;	
	//Preset valor posicao sequencia tempo homozenização	
	PRST_POSSEQ_TEMPO_HOMOGE AT %QW12488:INT;	

	//Contador da sequencia do Slurry Making
	CNT_SEQUENCIA_SLURRY AT %QW8004:INT;	
	
	//Preset Tempo de alarme descarga balanca de solido 1
	PRST_TEMPO_DESCARGA_BLS1 AT %QD12538:REAL;
	//Preset Tempo de alarme descarga balanca de solido 2		
	PRST_TEMPO_DESCARGA_BLS2 AT %QD12542:REAL;		
	//Preset Tempo de alarme descarga balanca de solido 3
	PRST_TEMPO_DESCARGA_BLS3 AT %QD12546:REAL;		
	//Preset Tempo de alarme descarga balanca de solido 4
	PRST_TEMPO_DESCARGA_BLS4 AT %QD12550:REAL;		
	//Preset Tempo de alarme descarga balanca de solido 5
	PRST_TEMPO_DESCARGA_BLS5 AT %QD12554:REAL;	
	//Preset Tempo de alarme descarga balanca de liquido 1	
	PRST_TEMPO_DESCARGA_BLL1 AT %QD12558:REAL;		
	//Preset Tempo de alarme descarga balanca de liquido 2
	PRST_TEMPO_DESCARGA_BLL2 AT %QD12562:REAL;	
	//Preset Tempo de alarme descarga balanca de liquido 3	
	PRST_TEMPO_DESCARGA_BLL3 AT %QD12566:REAL;	
	//Preset Tempo de alarme descarga balanca de liquido 4	
	PRST_TEMPO_DESCARGA_BLL4 AT %QD12570:REAL;
	//Preset Tempo de reação
	PRST_TEMPO_REACAO AT %QD12526:REAL;		
	//Preset tempo Hidratação	
	PRST_TEMPO_HIDRATACAO AT %QD12530:REAL;		
	//Preset tempo homogenizacao
	PRST_TEMPO_HOMOGENIZACAO AT %QD12534:REAL;

	//Preset Temperatura minima MXP
	PRST_TEMPE_MIN_MXP AT %QD12578:REAL;	
	//Preset Temperatura maxima MXP	
	PRST_TEMPE_MAX_MXP AT %QD12582:REAL;
	//Preset Temperatura alarme MXP		
	PRST_TEMPE_ALAR_MXP AT %QD12586:REAL;		
	
	//Contador Batelada
	LEITURA_BATELADA_ATUAL AT %QD13132:REAL;
	//Preset quantidade de bateladas		
	PRST_QNT_BATELADAS AT %QD12602:REAL;		
	
	//Preset Inicio escala Engenharia BLS1
	PRST_INI_ESCA_ENG_BLS1 AT %QD13400:REAL;		
	//Preset Inicio escala Engenharia BLS2
	PRST_INI_ESCA_ENG_BLS2 AT %QD13404:REAL;		
	//Preset Inicio escala Engenharia BLS3
	PRST_INI_ESCA_ENG_BLS3 AT %QD13408:REAL;		
	//Preset Inicio escala Engenharia BLS4
	PRST_INI_ESCA_ENG_BLS4 AT %QD13412:REAL;		
	//Preset Inicio escala Engenharia BLS5
	PRST_INI_ESCA_ENG_BLS5 AT %QD13416:REAL;		
	//Preset Inicio escala Engenharia BLL1
	PRST_INI_ESCA_ENG_BLL1 AT %QD13420:REAL;		
	//Preset Inicio escala Engenharia BLL2
	PRST_INI_ESCA_ENG_BLL2 AT %QD13424:REAL;		
	//Preset Inicio escala Engenharia BLL3
	PRST_INI_ESCA_ENG_BLL3 AT %QD13428:REAL;		
	//Preset Inicio escala Engenharia BLL4
	PRST_INI_ESCA_ENG_BLL4 AT %QD13432:REAL;		
	//Preset Fim escala Engenharia BLS1
	PRST_FIM_ESCA_ENG_BLS1 AT %QD13436:REAL;		
	//Preset Fim escala Engenharia BLS2
	PRST_FIM_ESCA_ENG_BLS2 AT %QD13440:REAL;		
	//Preset Fim escala Engenharia BLS3
	PRST_FIM_ESCA_ENG_BLS3 AT %QD13444:REAL;		
	//Preset Fim escala Engenharia BLS4
	PRST_FIM_ESCA_ENG_BLS4 AT %QD13448:REAL;		
	//Preset Fim escala Engenharia BLS5
	PRST_FIM_ESCA_ENG_BLS5 AT %QD13452:REAL;		
	//Preset Fim escala Engenharia BLL1
	PRST_FIM_ESCA_ENG_BLL1 AT %QD13456:REAL;		
	//Preset Fim escala Engenharia BLL2
	PRST_FIM_ESCA_ENG_BLL2 AT %QD13460:REAL;		
	//Preset Fim escala Engenharia BLL3
	PRST_FIM_ESCA_ENG_BLL3 AT %QD13464:REAL;		
	//Preset Fim escala Engenharia BLL4
	PRST_FIM_ESCA_ENG_BLL4 AT %QD13468:REAL;		
	//Preset Inicio escala KG BLS1
	PRST_INI_ESCA_KG_BLS1 AT %QD13472:REAL;		
	//Preset Inicio escala KG BLS2
	PRST_INI_ESCA_KG_BLS2 AT %QD13476:REAL;		
	//Preset Inicio escala KG BLS3
	PRST_INI_ESCA_KG_BLS3 AT %QD13480:REAL;		
	//Preset Inicio escala KG BLS4
	PRST_INI_ESCA_KG_BLS4 AT %QD13484:REAL;		
	//Preset Inicio escala KG BLS5
	PRST_INI_ESCA_KG_BLS5 AT %QD13488:REAL;		
	//Preset Inicio escala KG BLL1
	PRST_INI_ESCA_KG_BLL1 AT %QD13492:REAL;		
	//Preset Inicio escala KG BLL2
	PRST_INI_ESCA_KG_BLL2 AT %QD13496:REAL;		
	//Preset Inicio escala KG BLL3
	PRST_INI_ESCA_KG_BLL3 AT %QD13500:REAL;		
	//Preset Inicio escala KG BLL4
	PRST_INI_ESCA_KG_BLL4 AT %QD13504:REAL;		
	//Preset Fim escala KG BLS1
	PRST_FIM_ESCA_KG_BLS1 AT %QD13508:REAL;		
	//Preset Fim escala KG BLS2
	PRST_FIM_ESCA_KG_BLS2 AT %QD13512:REAL;		
	//Preset Fim escala KG BLS3
	PRST_FIM_ESCA_KG_BLS3 AT %QD13516:REAL;		
	//Preset Fim escala KG BLS4
	PRST_FIM_ESCA_KG_BLS4 AT %QD13520:REAL;		
	//Preset Fim escala KG BLS5
	PRST_FIM_ESCA_KG_BLS5 AT %QD13524:REAL;		
	//Preset Fim escala KG BLL1
	PRST_FIM_ESCA_KG_BLL1 AT %QD13528:REAL;		
	//Preset Fim escala KG BLL2
	PRST_FIM_ESCA_KG_BLL2 AT %QD13532:REAL;		
	//Preset Fim escala KG BLL3
	PRST_FIM_ESCA_KG_BLL3 AT %QD13536:REAL;		
	//Preset Fim escala KG BLL4
	PRST_FIM_ESCA_KG_BLL4 AT %QD13540:REAL;		
	
	//Preset nivel minimo Misturador Principal
	PRST_NIVEL_MINIMO_MPX AT %QD13568:REAL;		
	//Velocidade Misturador principal
	VEL_MPX:REAL;
	//Contador Batelada Geral
	LEITURA_BATELADA_TOTAL AT %QD13188:REAL;		
  	
	//Peso REAL Gravado BLS1
	LEITURA_PESO_GRAVADO_BLS1 AT %QD13208:REAL;		
	//Peso Real Gravado BLS2
	LEITURA_PESO_GRAVADO_BLS2 AT %QD13212:REAL;		
	//Peso Real Gravado BLS3
	LEITURA_PESO_GRAVADO_BLS3 AT %QD13216:REAL;		
	//Peso Real Gravado BLS4
	LEITURA_PESO_GRAVADO_BLS4 AT %QD13220:REAL;		
	//Peso Real Gravado BLS5
	LEITURA_PESO_GRAVADO_BLS5 AT %QD13224:REAL;		
	//Peso Real Gravado BLL1
	LEITURA_PESO_GRAVADO_BLL1 AT %QD13228:REAL;		
	//Peso Real Gravado BLL2
	LEITURA_PESO_GRAVADO_BLL2 AT %QD13232:REAL;		
	//Peso Real Gravado BLL3
	LEITURA_PESO_GRAVADO_BLL3 AT %QD13236:REAL;		
	//Peso Real Gravado BLL4
	LEITURA_PESO_GRAVADO_BLL4 AT %QD13240:REAL;	
	//Peso REAL Gravado Agua	
	LEITURA_PESO_GRAVADO_AGUA AT %QD13248:REAL;		
	


	
END_VAR

// Device/Application/GVLTransferencia
VAR_GLOBAL
	// STATUS MOINHO 02
	ST_MH_02 AT %QW15112: INT;
	
	//boleanos
		
	//Botão liga Exaustor FM1
	BTS_EXFM1 AT	%QX3004.1	:BOOL;
	//Nivel minimo mexedor de espera
	NIVEL_MINIMO_MXE AT %QX3040.0:BOOL;
	//Botão liga Mexedor espera	 
	BTS_MXE	AT	%QX3003.1	:BOOL;
	//Botão liga Bomba de baixa	 
	BTS_BB	AT	%QX3003.4	:BOOL;
	//Botão liga Bomba de alta 1	 
	BTS_BA1	AT	%QX3003.5	:BOOL;
	//Botão liga Bomba de alta 2	 
	BTS_BA2	AT	%QX3003.6	:BOOL;
	//Botão liga Moinho 	 
	BTS_MH	AT	%QX3004.0	:BOOL;
	//Botão manual/automatico on/off Transferencia		
	BTS_MATRANS AT %QX3005.2:BOOL;
	//Botão Liga Valvula de retorno
	BTS_VLR AT %QX3005.4:BOOL;	
	//Botão liga bomba de transferencia
	BTS_BBTRANSF AT %QX3005.7:BOOL;
	//Pressão alta na linha de alta
	PRESSAO_ALTA_LINHA_ALTA:BOOL;


	
	//Registros uso interno
	
	//Velocidade bomba de baixa
	VEL_BB AT %QD13000:REAL;	
		//Velocidade bomba de alta 1
	VEL_ALT1 AT %QD13004:REAL;	
	//Velocidade bomba de alta 2	
	VEL_ALT2 AT %QD13008:REAL;	
	//Pressão linha de alta	
	LEITURA_PRES_LA AT %QD13068:REAL;	
	//Pressão linha de baixa	
	LEITURA_PRES_LB AT %QD13072:REAL;	
	//Nivel Mexedor  de espera	
	LEITURA_NI_MXESPE AT %QD13080:REAL;		
	//Leitura Velocidade bomba de alta 1
	LEITURA_VEL_ALT1 AT %QD13084:REAL;	
	//Leitura Velocidade bomba de alta 2	
	LEITURA_VEL_ALT2 AT %QD13088:REAL;		
	//Nivel de religamento da bomba de transferencia
	NIVEL_RELIGAMENTO_BT:REAL;




END_VAR

//Supervisorio
VAR_GLOBAL PERSISTENT
	
	//Preset Pressão bomba de baixa
	PRST_PRESS_BB AT %QD12574:REAL;	
	//Velocidade da bomba de baixa
	PRST_VEL_BB AT %QD12408:REAL;	
	//Velocidade da bomba de alta 1
	PRST_VEL_BA1 AT %QD12412:REAL;
	//Velocidade da bomba de alta 2
	PRST_VEL_BA2 AT %QD12416:REAL;
	//Preset nivel minimo Misturador de espera
	PRST_MIN_MISTESPERA AT %QD12590:REAL;	
	//Preset nivel maximo Misturador de espera	
	PRST_MAX_MISTESPERA AT %QD12594:REAL;
	//Tolerancia nivel misturador de espera religamento bomba transferencia em %
	PRST_TOL_NIVEL_MXESP_BT AT %QD12598:REAL;	
	//Preset maximo pressao linha de alta
	PRST_MAX_PRESSAO_BA AT %QD12606:REAL;	
	//Preset pressao libera sopro	
	PRST_PRESSAO_LIB_SOPRO AT %QD12610:REAL;	
	//Preset pressao libera reciclo	
	PRST_PRESSAO_LIB_RECICLO AT %QD12614:REAL;		

	
	//Botão Habilita Bomba de alta 1
	BTS_HAB_BA1 AT %QX3017.7:BOOL;	
	//Botão habilita bomba de alta 2	
	BTS_HAB_BA2 AT %QX3018.0:BOOL;		

		


END_VAR

// Device/Application/GVLTorre
VAR_GLOBAL
	//boleanos
	
	//Botão manual/automatico off/on SprayDrying
	BTS_SPRAYDRYING AT %QX3005.1:BOOL;
	//Botão liga exaustor da torre (125 cv)
	BTS_EXTORRE AT %QX3006.4:BOOL;
	//Botão liga ventilador do queimador
	BTS_VENTIQUEIMADOR AT %QX3006.5:BOOL;
	//Botão liga Esteira TC02	 
	BTS_ESTTC02 AT	%QX3004.5	:BOOL;
	//Botão liga Air Lifit em 100%	 
	BTS_VELAIRLF AT	%QX3004.6	:BOOL;
	//Sopro liberado
	SOPRO_LIBERADO AT %QX3040.1:BOOL;	
	//Botão libera sem PH
	BTS_LIBERA_SEMPH AT %QX3018.1:BOOL;	
	//Botão Dumper torre off – atm/ on-torre	
	BTS_DUMPER_TORRE AT %QX3018.2:BOOL;	
	//Botão Partida queimador remota	
	BTS_PARTIDAQUEIMADOR_REM AT %QX3018.3:BOOL;	
	//Sopro sem PH	
	SOPRO_SEM_PH AT %QX3040.4:BOOL;
	//Dosador Torre habilitado		
	DSATORRE_HAB AT %QX3040.5:BOOL;		


	//libera Dumper
	LIB_DUMPER:BOOL;	
	
	//Registros uso interno
	
	//Velocidade exaustor da torre (125 cv) 0-100%
	VEL_EXTORRE AT %QD13012:REAL;
	//Velocidade ventilador queimador 0-100%
	VEL_VENTQUEIMADOR AT %QD13016:REAL;	
	//Leitura Pressão Torre	
	LEITURA_PRES_TORRE AT %QD13092:REAL;	
	//Base soprada na torre
	LEITURA_BASE_SOP_TORRE AT %QD13136:REAL;
	//Número de Jatos abertos
	QTD_JATOS AT %QD13308:REAL;	
	//Realizar gravação das pressoes e temperatura	
	GRAVAR_DADOS_ANALOGICAS AT %QD13252:REAL;
	//Preset Reset Leitura variaveis analogicas
	PRST_RESET_LEITURA_ANALOICA AT %QD13560:REAL;	
	
	//Roby - Alterado em 23/02/2021
	// Valor de medição de umidade no supervisório
	VALOR_MEDICAO_UMIDADE AT %QW13296:REAL;
	
	//Roby - Alterado em 23/02/2021==========================INÍCO==========================
	// Valor de pressão da tubulação do óleo BPF que alimenta a caldeira
	PRESS_OLEO_BPF AT %QW13300:REAL;
	//Roby - Alterado em 23/02/2021==========================FIM==========================
	
	
END_VAR


// Supervisório
VAR_GLOBAL PERSISTENT
	
	//Velocidade do exaustor da torre (125 cv)
	PRST_VEL_EXTORRE AT %QD12428:REAL;	
	//velocidade ventilador queimador
	PRST_VEL_VENTIQUEIMADOR AT %QD12432:REAL;
	//preset vazao oleo queimador
	PRST_OLEO_QUEIMADOR AT %QD12452:REAL;
	//Preset percentual sulfato torre
	PRST_PERC_SULFATO_DSTORRE AT %QD12814:REAL;	
	//Preset Us dosador torre	
	PRST_US_DSTORRE AT %QD12818:REAL;
	//Preset Ub dosador torre		
	PRST_UB_DSTORRE AT %QD12822:REAL;
	//Preset ds dosador torre	
	PRST_DS_DSTORRE AT %QD12826:REAL;		
	//Preset temperatura seguranca torre
	PRST_SEGURANCA_TORRE AT %QD13552:REAL;	
	// Preset Relacao po base	
	PRST_RELACAO_PO_BASE AT %QD13564:REAL;		



END_VAR

// Device/Application/GVLPH
VAR_GLOBAL
	
		
	//Botão liga Exaustor FM2 	 
	BTS_EXFM2 AT	%QX3004.2	:BOOL;
	//Botão liga ventilador FM2 	
	BTS_EXVFM2 AT	%QX3004.3	:BOOL;
	//Botão liga ventilador do Fluidizador
	BTS_VENTIFLUIDIZADOR AT %QX3006.6:BOOL;	
	//Botão manual/automatico off/on PH 1
	BTS_MAPH1 AT %QX3006.7:BOOL;		
	//Botão liga bomba alimentação de oleo
	BTS_BALIOLEO AT %QX3007.0:BOOL;
	//Botão liga Esteira TC8	
	BTS_ESTTC8 AT %QX3007.1:BOOL;	
	//Botão liga Esteira TC8 reversão
	BTS_ESTTC8REVER AT %QX3007.2:BOOL;	
	//Botão liga bomba de perfume 1	
	BTS_BP1 AT %QX3007.3:BOOL;	
	//Botão liga bomba de perfume 2	
	BTS_BP2 AT %QX3007.4:BOOL;
	//Botão manual/automatico off/on PH 2
	BTS_MAPH2 AT %QX3007.5:BOOL;
	//Botão liga Peneiras
	BTS_PNS AT %QX3007.6:BOOL;	
	//Botão liga esteira saida da torre	
	BTS_ESTSATORRE AT %QX3007.7:BOOL;	
	//Botão liga esteira TC13
	BTS_ESTTC13 AT %QX3008.0:BOOL;	
	//Botão liga Esteira TC3 Dry Mix	
	BTS_TC3	AT	%QX3004.4	:BOOL;
	//Botão liga Elevador 2	
	BTS_EL2	AT	%QX3004.7	:BOOL;	
	//Botão liga Dosador 6 – linha 1		
	BTS_DS6 AT %QX3008.6:BOOL;	
	//Botão liga Elevador 4
	BTS_EL4 AT %QX3018.4:BOOL;	
	//Botão habilita sopragem sem PH	
	BTS_HAB_SOPRO_SEMPH AT %QX3018.5:BOOL;	
	//Botão liga filtro manga 2
	BTS_FILTM2 AT %QX3018.6:BOOL;
	//Botão Reset totalizador dos Dosadores Schenck
	BTS_RESET_TOTAL_SCHENCK AT %QX3020.1:BOOL;		
		


	//Desliga carregamento fluidizador 1 por peso maximo
	NIVEL_MAXIMO_FLUID1 AT %QX3040.2:BOOL;	
	//Desliga carregamento fluidizador 2 por peso maximo
	NIVEL_MAXIMO_FLUID2 AT %QX3040.3:BOOL;		
	//Botão liga filtro manga 1
	BTS_FILTM1 AT %QX3006.3:BOOL;
	//Desliga fluidizador 1
	DESLIGA_FLUIDIZADOR1:BOOL;
	//Desliga fluidizador 2
	DESLIGA_FLUIDIZADOR2:BOOL;
	//Liga filtr manga 1
	LIGA_FTM1:BOOL;
	//Liga filtr manga 2
	LIGA_FTM2:BOOL;
	
	//Velocidade ventilador fluidizador 0-100%
	VEL_VENTFLUIDIZADOR AT %QD13020:REAL;
	//Velocidade bomba perfume 1 0- 99.99hz (escala aberta +)
	VEL_BP1 AT %QD13024:REAL;	
	//Velocidade bomba perfume 2 0- 99.99hz (escala aberta +)
	VEL_BP2 AT %QD13028:REAL;
	//Leitura peso fluidizador 1
	LEITURA_PESO_FLUI1 AT %QD13096:REAL;
	//Leitura peso fluidizador 2		
	LEITURA_PESO_FLUI2 AT %QD13100:REAL;		
	//leitura velocidade DSA1	
	LEITURA_VELDSA1 AT %QD13124:REAL;
	//Velocidade dosdor 6
	VEL_DSA6 AT %QD8000:REAL;	
	//Leitura Velocidade Dosador 6
	LEITURA_VEL_DSA6 AT %QD13128:REAL;	
	//Leitura velocidade BBP1
	LEITURA_VEL_BBP1 AT %QD13140:REAL;	
	//Leitura velocidade BBP2	
	LEITURA_VEL_BBP2 AT %QD13144:REAL;		
	//Velocidade PH1 em Kg pelo PID em Auto
	VELOCIDADE_PH1_AUTO AT %QD13192:REAL;
	//Velocidade PH2 em Kg pelo PID em Auto
	VELOCIDADE_PH2_AUTO AT %QD13196:REAL;
	
	
	// Vazao Volumetrica Real BBP01 (dm³/h)
	VAZAO_VOLUMETRICA_REAL_BBP01: REAL;
	// Vazao Volumetrica Real BBP02 (dm³/h)
	VAZAO_VOLUMETRICA_REAL_BBP02: REAL;
	// TOTALIZADOR 1 BBP01
	TOTALIZADOR1_BBP01 AT %QD13260: REAL;
	// TOTALIZADOR 2 BBP01
	TOTALIZADOR2_BBP01 AT %QD13256: REAL;
	// TOTALIZADOR 3 BBP01
	TOTALIZADOR3_BBP01 AT %QD13268: REAL;
	// TOTALIZADOR 1  BBP02
	TOTALIZADOR1_BBP02 AT %QD13272: REAL;
	// TOTALIZADOR 3 BBP02
	TOTALIZADOR3_BBP02 AT %QD13280: REAL;
	// Zera Totalizador 1 BBP01
	BTS_ZERA_TOTALIZADOR1_BBP01 AT %QX3020.2: BOOL;
	// Totalizador 2 da BBP01
	TOTALIZADOR2_BBP02 AT %QD13276: REAL;
	// Status dosador 07 habilitado
	DS07_HAB: BOOL;
END_VAR

// Supervisório
VAR_GLOBAL PERSISTENT
			
	//Velocidade ventilador fluidizador 0-100%
	PRST_VEL_VENTIFLUIDIZADOR AT %QD12436:REAL;	
		
	
	//Preset Peso Maximo Fluidizador 1	
	PRST_PESO_MAX_FLUID1 AT %QD12618:REAL;
	//Preset Peso Minimo Fluidizador 1
	PRST_PESO_MIN_FLUID1 AT %QD12622:REAL;
	//Preset Peso Maximo Fluidizador 2
	PRST_PESO_MAX_FLUID2 AT %QD12626:REAL;
	//Preset Peso Minimo Fluidizador 2
	PRST_PESO_MIN_FLUID2 AT %QD12630:REAL;
	//Preset Peso Fluidizador
	PRST_PESO_FLUIDIZADOR1 AT %QD12702:REAL;	
	//Preset Peso Fluidizador	
	PRST_PESO_FLUIDIZADOR2 AT %QD12706:REAL;		
	//Preset Velocidade PH1 Manual
	PRST_VEL_PH1_MANUAL AT %QD12694:REAL;	
	//Preset Velocidade PH2 Manual	
	PRST_VEL_PH2_MANUAL AT %QD12698:REAL;	
	//Producao PH1 De	
	PRST_PRODUCAO_PH1_DE AT %QD12710:REAL;	
	//Producao PH1 A	
	PRST_PRODUCAO_PH1_A AT %QD12714:REAL;		
	//Producao PH2 De
	PRST_PRODUCAO_PH2_DE AT %QD12718:REAL;	
	//Producao PH2 A	
	PRST_PRODUCAO_PH2_A AT %QD12722:REAL;	

	//Velocidade bomba perfume 1	
	PRST_VEL_BPF1 AT %QD12440:REAL;	
	//Velocidade bomba perfume 2	
	PRST_VEL_BPF2 AT %QD12444:REAL;	
	//Preset velocidade DS2 Schenck calculado	
	PRST_VEL_DS2 AT %QD12726:REAL;	
	//Preset velocidade DS3 Schenck calculado	
	PRST_VEL_DS3 AT %QD12730:REAL;
	//Preset velocidade DS4 Schenck calculado		
	PRST_VEL_DS4 AT %QD12734:REAL;	
	//Preset velocidade DS5 Schenck calculado	
	PRST_VEL_DS5 AT %QD12738:REAL;	
	//Preset velocidade DS7 Schenck calculado	
	PRST_VEL_DS7 AT %QD12742:REAL;		
	//Preset velocidade DS8 Schenck calculado
	PRST_VEL_DS8 AT %QD12746:REAL;	
	//Preset velocidade DS9 Schenck calculado	
	PRST_VEL_DS9 AT %QD12750:REAL;	
	//Preset velocidade DS10 Schenck calculado	
	PRST_VEL_DS10 AT %QD12754:REAL;	
	//Preset velocidade DS11 Schenck calculado	
	PRST_VEL_DS11 AT %QD12758:REAL;		
	//Preset velocidade DS12 Schenck calculado
	PRST_VEL_DS12 AT %QD12762:REAL;
	// Preset velocidade DS14 Schenck calculado
	PRST_VEL_DS14 AT %QD13576:REAL;
	//Preset velocidade DSTORRE Schenck calculado		
	PRST_VEL_DSTORRE AT %QD12766:REAL;	
	//Preset velocidade DS1 Schenck calculado	
	PRST_VEL_DS1 AT %QD12770:REAL;	
	//Velocidade Dosador 6
	PRST_VEL_DS6 AT %QD12774:REAL;	
		

	
	//Preset Percentual velocidade dosagem dosador Po base 1
	PRST_PERC_DOSA_PB01 AT %QD12634:REAL;
	//Preset Percentual velocidade dosagem dosador Po base 11		
	PRST_PERC_DOSA_PB11 AT %QD12638:REAL;	
	//Preset Percentual velocidade dosagem Bomba perfume 1	
	PRST_PERC_DOSA_BBP01 AT %QD12642:REAL;		
	//Preset Percentual velocidade dosagem Bomba perfume 2
	PRST_PERC_DOSA_BBP02 AT %QD12646:REAL;	
	//Preset Percentual velocidade dosagem Dosador 2	
	PRST_PERC_DOSA_DS02 AT %QD12650:REAL;		
	//Preset Percentual velocidade dosagem Dosador 3
	PRST_PERC_DOSA_DS03 AT %QD12654:REAL;
	//Preset Percentual velocidade dosagem Dosador 4		
	PRST_PERC_DOSA_DS04 AT %QD12658:REAL;	
	//Preset Percentual velocidade dosagem Dosador 5	
	PRST_PERC_DOSA_DS05 AT %QD12662:REAL;		
	//Preset Percentual velocidade dosagem Dosador 6	
	PRST_PERC_DOSA_DS06 AT %QD12666:REAL;		
	//Preset Percentual velocidade dosagem Dosador 7
	PRST_PERC_DOSA_DS07 AT %QD12670:REAL;		
	//Preset Percentual velocidade dosagem Dosador 8
	PRST_PERC_DOSA_DS08 AT %QD12674:REAL;	
	//Preset Percentual velocidade dosagem Dosador 9	
	PRST_PERC_DOSA_DS09 AT %QD12678:REAL;
	//Preset Percentual velocidade dosagem Dosador 10		
	PRST_PERC_DOSA_DS10 AT %QD12682:REAL;		
	//Preset Percentual velocidade dosagem Dosador 12
	PRST_PERC_DOSA_DS12 AT %QD12686:REAL;		
	// Preset Percentual velocidade dosagem Dosador 14
	PRST_PERC_DOSA_DS14 AT %QD13572:REAL;		
	//Preset Percentual velocidade dosagem Dosador Torre
	PRST_PERC_DOSA_DSTORRE AT %QD12690:REAL;		
	
	//Preset Altura Dosador 6
	PRST_ALTURA_DS6 AT %QD12778:REAL;
	//Preset Largura Dosador 6		
	PRST_LARGURA_DS6 AT %QD12782:REAL;	
	//Preset Densidade Produto Dosador 6	
	PRST_DENSIDADE_DS6 AT %QD12786:REAL;		
	//Preset Constante A Dosador 6	
	PRST_CONSTANTE_A_DS6 AT %QD12790:REAL;
	//Preset Constante B Dosador 6
	PRST_CONSTANTE_B_DS6 AT %QD12794:REAL;
	//Preset Constante A BBP01
	PRST_CONSTANTE_A_BBP01 AT %QD12798:REAL;
	//Preset Constante B BBP01		
	PRST_CONSTANTE_B_BBP01 AT %QD12802:REAL;	
	//Preset Constante A BBP02	
	PRST_CONSTANTE_A_BBP02 AT %QD12806:REAL;	
	//Preset Constante B BBP02	
	PRST_CONSTANTE_B_BBP02 AT %QD12810:REAL;		
	// Velocidade programada da bomba de perfume 1 (kg/h)
	VEL_PROGRAMADA_BBP01 AT %QD13288: REAL;
	// Velocidade programada da bomba de perfume 2 (kg/h)
	VEL_PROGRAMADA_BBP02 AT %QD13292: REAL;


	//Quantidade dosado Bomba Perfume 1
	LEITURA_QTD_DOSADO_BPF1 AT %QD13200:REAL;
	//Quantidade dosado Bomba Perfume 2	
	LEITURA_QTD_DOSADO_BPF2 AT %QD13204:REAL;
	//Preset razão pulsos DO perfume bomba 1
	PRST_RAZAO_BPF1 AT %QD13544:REAL;	
	// Densidade relativa da BBP02, relação com a água
	MASSA_ESPECIFICA_BBP02 AT %QD13284: REAL;
	// Densidade relativa da BBP01, relação com a água
	MASSA_ESPECIFICA_BBP01 AT %QD13264: REAL;
	//Preset razão pulsos do perfume bomba 2	
	PRST_RAZAO_BPF2 AT %QD13548:REAL;		

	
END_VAR

// Device/Application/GVLTemperaturas
VAR_GLOBAL
	//Temperatura do vapor misturador
	TEMP_VAPOR AT %QD13104:REAL;
	// Temperatura da torre tipok
	TEMP_TORRE AT %QD13108:REAL;
	//Temperatura do queimador para torre
	TEMP_QUEIMATORRE AT %QD13112:REAL;
	//Temperatura do queimador para atmosfera
	TEMP_QUEIMAATM AT %QD13116:REAL;
	// Temperatura da torre PT100
	TEMPERATURA_TORRE AT %QD13120: REAL;
END_VAR

// Device/Application/GVLSCHENCK
VAR_GLOBAL
		
	//Liga Dosador 1 - linha 1
	LIGA_DS1:BOOL;
	//Liga Dosador 2 - linha 1
	LIGA_DS2:BOOL;
	//Liga Dosador 3 - linha 1
	LIGA_DS3:BOOL;
	//Liga Dosador 4 - linha 1
	LIGA_DS4:BOOL;
	//Liga Dosador 5 - linha 1
	LIGA_DS5:BOOL;
	//Liga Dosador 7 - linha 1
	LIGA_DS7:BOOL;
	//Liga Dosador 8 - linha 1
	LIGA_DS8:BOOL;
	//Liga Dosador 9 - linha 1
	LIGA_DS9:BOOL;
	//Liga Dosador 10 - linha 1
	LIGA_DS10:BOOL;
	//Liga Dosador 11 - linha 1
	LIGA_DS11:BOOL;
	//Liga Dosador 12 - linha 1
	LIGA_DS12:BOOL;
	// Liga Dosador 14 - linha 1
	LIGA_DS14: BOOL;
	//Liga Dosador Torre - linha 1
	LIGA_DSTORRE:BOOL;
	
			
	
	//Botão liga Dosador Gravimetrico 1 DEA-600 D-2B linha 1
	BTS_DS1 AT %QX3008.1:BOOL;
	//Botão comando limpa eventos - dosador Gravimetrico 1 DEA-600 D-2B linha 1	
	BTS_LIMPEVE_DS1 AT %QX3010.0:BOOL;			
	//Botão comando zera totalizador 1 - dosador Gravimetrico 1 DEA-600 D-2B linha 1	
	BTS_ZERATOTAL1_DS1 AT %QX3010.3:BOOL;		
	//Botão comando zera totalizador 2 - dosador Gravimetrico 1 DEA-600 D-2B linha 1	
	BTS_ZERATOTAL2_DS1 AT %QX3010.4:BOOL;
	
	
	//Botão liga Dosador Gravimetrico 2 DEA-300 D-4B linha 1
	BTS_DS2 AT %QX3008.2:BOOL;	
	//Botão comando limpa eventos - dosador Gravimetrico 2 DEA-300 D-4B linha 1	
	BTS_LIMPEVE_DS2 AT %QX3010.5:BOOL;				
	//Botão comando zera totalizador 1 - dosador Gravimetrico 2 DEA-300 D-4B linha 1	
	BTS_ZERATOTAL1_DS2 AT %QX3011.0:BOOL;		
	//Botão comando zera totalizador 2 - dosador Gravimetrico 2 DEA-300 D-4B linha 1	
	BTS_ZERATOTAL2_DS2 AT %QX3011.1:BOOL;	
		

	//Botão liga Dosador Gravimetrico 3 DEA-300 D-3B linha 1	
	BTS_DS3 AT %QX3008.3:BOOL;	
	//Botão comando zera eventos - dosador Gravimetrico 3 DEA-300 D-3B linha 1		
	BTS_LIMPEVE_DS3 AT %QX3011.2:BOOL;				
	//Botão comando zera totalizador 1 - dosador Gravimetrico 3 DEA-300 D-3B linha 1	
	BTS_ZERATOTAL1_DS3 AT %QX3011.5:BOOL;		
	//Botão comando zera totalizador 2 - dosador Gravimetrico 3 DEA-300 D-3B linha 1	
	BTS_ZERATOTAL2_DS3 AT %QX3011.6:BOOL;	
	
	
	//Botão liga Dosador Gravimetrico 4 MECHATRON D-6B linha 1
	BTS_DS4 AT %QX3008.4:BOOL;
	//Botão comando zera evento - dosador Gravimetrico 4 MECHATRON D-6B linha 1	
	BTS_LIMPEVE_DS4 AT %QX3011.7:BOOL;		
	//Botão comando zera totalizador 1 - dosador Gravimetrico 4 MECHATRON D-6B linha 1	
	BTS_ZERATOTAL1_DS4 AT %QX3012.2:BOOL;		
	//Botão comando zera totalizador 2 - dosador Gravimetrico 4 MECHATRON D-6B linha 1	
	BTS_ZERATOTAL2_DS4 AT %QX3012.3	:BOOL;	

	
	//Botão liga Dosador Gravimetrico 5 MECHATRON D-7B linha 1
	BTS_DS5 AT %QX3008.5:BOOL;	
	//Botão comando zera eventos - dosador Gravimetrico 5 MECHATRON D-7B linha 1	
	BTS_LIMPEVE_DS5 AT %QX3012.4:BOOL;		
	//Botão comando zera totalizador 1 - dosador Gravimetrico 5 MECHATRON D-7B linha 1	
	BTS_ZERATOTAL1_DS5 AT %QX3012.7:BOOL;		
	//Botão comando zera totalizador 2 - dosador Gravimetrico 5 MECHATRON D-7B linha 1	
	BTS_ZERATOTAL2_DS5 AT %QX3013.0 :BOOL;		
	
	
	//Botão liga Dosador Gravimetrico 7 MECHATRON D-5A linha 2
	BTS_DS7 AT %QX3008.7:BOOL;	
	//Botão comando zera eventos - dosador Gravimetrico 7 MECHATRON D-5A linha 2
	BTS_LIMPEVE_DS7 AT %QX3013.1:BOOL;		
	//Botão comando zera totalizador 1 - dosador Gravimetrico 7 MECHATRON D-5A linha 2
	BTS_ZERATOTAL1_DS7 AT %QX3013.4:BOOL;
	//Botão comando zera totalizador 2 - dosador Gravimetrico 7 MECHATRON D-5A linha 2
	BTS_ZERATOTAL2_DS7 AT %QX3013.5:BOOL;

		
	//Botão liga Dosador Gravimetrico 8 MECHATRON D-7A linha 2	
	BTS_DS8 AT %QX3009.0:BOOL;
	//Botão comando zera eventos - dosador Gravimetrico 8 MECHATRON D-7A linha 2
	BTS_LIMPEVE_DS8 AT %QX3013.6:BOOL;		
	//Botão comando zera totalizador 1 - dosador Gravimetrico 8 MECHATRON D-7A linha 2
	BTS_ZERATOTAL1_DS8 AT %QX3014.1:BOOL;
	//Botão comando zera totalizador 2 - dosador Gravimetrico 8 MECHATRON D-7A linha 2
	BTS_ZERATOTAL2_DS8 AT %QX3014.2:BOOL;
	

	//Botão liga Dosador Gravimetrico 9 MECHATRON D-6A linha 2		
	BTS_DS9 AT %QX3009.1:BOOL;
	//Botão comando zera eventos - dosador Gravimetrico 9 MECHATRON D-6A linha 2
	BTS_LIMPEVE_DS9 AT %QX3014.3:BOOL;		
	//Botão comando zera totalizador 1 - dosador Gravimetrico 9 MECHATRON D-6A linha 2
	BTS_ZERATOTAL1_DS9 AT %QX3014.6:BOOL;
	//Botão comando zera totalizador 2 - dosador Gravimetrico 9 MECHATRON D-6A linha 2
	BTS_ZERATOTAL2_DS9 AT %QX3014.7:BOOL;
	
	
	//Botão liga Dosador Gravimetrico 10 MECHATRON DEA-4A linha 2		
	BTS_DS10 AT %QX3009.2:BOOL;
	//Botão comando zera eventos - dosador Gravimetrico 10 MECHATRON DEA-4A linha 2
	BTS_LIMPEVE_DS10 AT %QX3015.0:BOOL;		
	//Botão comando zera totalizador 1 - dosador Gravimetrico 10 MECHATRON DEA-4A linha 2
	BTS_ZERATOTAL1_DS10 AT %QX3015.3:BOOL;	
	//Botão comando zera totalizador 2 - dosador Gravimetrico 10 MECHATRON DEA-4A linha 2
	BTS_ZERATOTAL2_DS10 AT %QX3015.4:BOOL;
	
		
	//Botão liga Dosador Gravimetrico 11 MECHATRON DEA-2A linha 2		
	BTS_DS11 AT %QX3009.3:BOOL;	
	//Botão comando zera eventos - dosador Gravimetrico 11 MECHATRON DEA-2A linha 2
	BTS_LIMPEVE_DS11 AT %QX3015.5:BOOL;		
	//Botão comando zera totalizador 1 - dosador Gravimetrico 11 MECHATRON DEA-2A linha 2
	BTS_ZERATOTAL1_DS11 AT %QX3016.0:BOOL;	
	//Botão comando zera totalizador 2 - dosador Gravimetrico 11 MECHATRON DEA-2A linha 2
	BTS_ZERATOTAL2_DS11 AT %QX3016.1:BOOL;


	//Botão liga Dosador Gravimetrico 12 MECHATRON DEA-3A linha 2	
	BTS_DS12 AT %QX3009.4:BOOL;	
	//Botão comando zera eventos - dosador Gravimetrico 12 MECHATRON DEA-3A linha 2
	BTS_LIMPEVE_DS12 AT %QX3016.2:BOOL;	
	//Botão comando zera totalizador 1 - dosador Gravimetrico 12 MECHATRON DEA-3A linha 2
	BTS_ZERATOTAL1_DS12 AT %QX3016.5:BOOL;	
	//Botão comando zera totalizador 2 - dosador Gravimetrico 12 MECHATRON DEA-3A linha 2
	BTS_ZERATOTAL2_DS12 AT %QX3016.6:BOOL;
	// Botão liga Dosador Gravimetrico 14 MECHATRON 
	BTS_DS14 AT %QX3022.0: BOOL;
	// Botão comando zera eventos - dosador Gravimetrico 14
	BTS_LIMPEVE_DS14 AT %QX3022.2: BOOL;
	// Botão comando zera totalizador 1 - dosador Gravimetrico 14 
	BTS_ZERATOTAL1_DS14 AT %QX3022.4: BOOL;
	// Botão comando zera totalizador 2 - dosador Gravimetrico 14 
	BTS_ZERATOTAL2_DS14 AT %QX3022.5: BOOL;
	
	
	//Botão liga Dosador TORRE	MECHATRON DEA-D1
	BTS_DSTORRE AT %QX3009.5:BOOL;	
	//Botão comando zera eventos - dosador Sulfato torre  MECHATRON DEA-D1
	BTS_LIMPEVE_DSTORRE AT %QX3016.7:BOOL;		
	//Botão comando zera totalizador 1 - dosador Sulfato torre  MECHATRON DEA-D1
	BTS_ZERATOTAL1_DSTORRE AT %QX3017.2:BOOL;
	//Botão comando zera totalizador 2 - dosador Sulfato torre  MECHATRON DEA-D1
	BTS_ZERATOTAL2_DSTORRE AT %QX3017.3:BOOL;

		
	//Bits comando Dosador Gravimetrico 1 DEA-600 D-2B linha 1
	COMMAND_DSA1 AT %QW15000:WORD;
	//Bits comando Dosador Gravimetrico 2 DEA-300 D-4B linha 1
	COMMAND_DSA2 AT %QW15002:WORD;
	//Bits comando Dosador Gravimetrico 3 DEA-300 D-3B linha 1
	COMMAND_DSA3 AT %QW15004:WORD;
	//Bits comando Dosador Gravimetrico 4 MECHATRON D-6B linha 1
	COMMAND_DSA4 AT %QW15006:WORD;
	//Bits comando Dosador Gravimetrico 5 MECHATRON D-7B linha 1
	COMMAND_DSA5 AT %QW15008:WORD;
	//Bits comando Dosador Gravimetrico 7 MECHATRON D-5A linha 2
	COMMAND_DSA7 AT %QW15010:WORD;
	//Bits comando Dosador Gravimetrico 8 MECHATRON D-7A linha 2	
	COMMAND_DSA8 AT %QW15012:WORD;
	//Bits comando Dosador Gravimetrico 9 MECHATRON D-6A linha 2
	COMMAND_DSA9 AT %QW15014:WORD;
	//Bits comando Dosador Gravimetrico 10 MECHATRON DEA-4A linha 2
	COMMAND_DSA10 AT %QW15016:WORD;
	//Bits comando Dosador Gravimetrico 11 MECHATRON DEA-2A linha 2
	COMMAND_DSA11 AT %QW15018:WORD;
	//Bits comando Dosador Gravimetrico 12 MECHATRON DEA-3A linha 2
	COMMAND_DSA12 AT %QW15020:WORD;
	// Bits comando Dosador Gravimetrico 14
	COMMAND_DSA14 AT %QW15024: WORD;
	//Bits comando Dosador TORRE MECHATRON DEA-D1
	COMMAND_DSATORRE AT %QW15022:WORD;
	
	
	//Bits status Dosador Gravimetrico 1 DEA-600 D-2B linha 1
	STATUS_DSA1 AT %IW15030:WORD;
	//Bits status Dosador Gravimetrico 2 DEA-300 D-4B linha 1
	STATUS_DSA2 AT %IW15032:WORD;
	//Bits status Dosador Gravimetrico 3 DEA-300 D-3B linha 1
	STATUS_DSA3 AT %IW15034:WORD;
	//Bits status Dosador Gravimetrico 4 MECHATRON D-6B linha 1
	STATUS_DSA4 AT %IW15036:WORD;
	//Bits status Dosador Gravimetrico 5 MECHATRON D-7B linha 1
	STATUS_DSA5 AT %IW15038:WORD;
	//Bits status Dosador Gravimetrico 7 MECHATRON D-5A linha 2
	STATUS_DSA7 AT %IW15040:WORD;
	//Bits status Dosador Gravimetrico 8 MECHATRON D-7A linha 2	
	STATUS_DSA8 AT %IW15042:WORD;
	//Bits status Dosador Gravimetrico 9 MECHATRON D-6A linha 2
	STATUS_DSA9 AT %IW15044:WORD;
	//Bits status Dosador Gravimetrico 10 MECHATRON DEA-4A linha 2
	STATUS_DSA10 AT %IW15046:WORD;
	//Bits status Dosador Gravimetrico 11 MECHATRON DEA-2A linha 2
	STATUS_DSA11 AT %IW15048:WORD;
	//Bits status Dosador Gravimetrico 12 MECHATRON DEA-3A linha 2
	STATUS_DSA12 AT %IW15050:WORD;
	// Bits status Dosador Gravimetrico 14
	STATUS_DSA14 AT %IW15054: WORD;
	//Bits status Dosador TORRE MECHATRON DEA-D1
	STATUS_DSATORRE AT %IW15052:WORD;
	
	//Bits status Alarme System Message Dosador Gravimetrico 1 DEA-600 D-2B linha 1
	STATUS_ALARM_SYSTEM_DSA1 AT %IW15360:WORD;
	//Bits status Alarme System Dosador Gravimetrico 2 DEA-300 D-4B linha 1
	STATUS_ALARM_SYSTEM_DSA2 AT %IW15362:WORD;
	//Bits status Alarme System Dosador Gravimetrico 3 DEA-300 D-3B linha 1
	STATUS_ALARM_SYSTEM_DSA3 AT %IW15364:WORD;
	//Bits status Alarme System Dosador Gravimetrico 4 MECHATRON D-6B linha 1
	STATUS_ALARM_SYSTEM_DSA4 AT %IW15366:WORD;
	//Bits comando Alarme System Dosador Gravimetrico 5 MECHATRON D-7B linha 1
	STATUS_ALARM_SYSTEM_DSA5 AT %IW15368: WORD;
	//Bits status Alarme System Dosador Gravimetrico 7 MECHATRON D-5A linha 2
	STATUS_ALARM_SYSTEM_DSA7 AT %IW15370:WORD;
	//Bits status Alarme System Dosador Gravimetrico 8 MECHATRON D-7A linha 2	
	STATUS_ALARM_SYSTEM_DSA8 AT %IW15372:WORD;
	//Bits status Alarme System Dosador Gravimetrico 9 MECHATRON D-6A linha 2
	STATUS_ALARM_SYSTEM_DSA9 AT %IW15374:WORD;
	//Bits status Alarme System Dosador Gravimetrico 10 MECHATRON DEA-4A linha 2
	STATUS_ALARM_SYSTEM_DSA10 AT %IW15376:WORD;
	//Bits status Alarme System Dosador Gravimetrico 11 MECHATRON DEA-2A linha 2
	STATUS_ALARM_SYSTEM_DSA11 AT %IW15378:WORD;
	//Bits status Alarme System Dosador Gravimetrico 12 MECHATRON DEA-3A linha 2
	STATUS_ALARM_SYSTEM_DSA12 AT %IW15380:WORD;
	// Bits status Alarme System Dosador Gravimetrico 14
	STATUS_ALARM_SYSTEM_DSA14 AT %IW15384: WORD;
	//Bits status Alarme System Dosador TORRE MECHATRON DEA-D1
	STATUS_ALARM_SYSTEM_DSATORRE AT %IW15382:WORD;
	
	//Bits status Alarme Sequence Monitoring Dosador Gravimetrico 1 DEA-600 D-2B linha 1
	STATUS_ALARM_SEQUENCE_DSA1 AT %IW15384:WORD;
	//Bits status Alarme Sequence Monitoring Dosador Gravimetrico 2 DEA-300 D-4B linha 1
	STATUS_ALARM_SEQUENCE_DSA2 AT %IW15386:WORD;
	//Bits status Alarme Sequence Monitoring Dosador Gravimetrico 3 DEA-300 D-3B linha 1
	STATUS_ALARM_SEQUENCE_DSA3 AT %IW15388:WORD;
	//Bits status Alarme Sequence Monitoring Dosador Gravimetrico 4 MECHATRON D-6B linha 1
	STATUS_ALARM_SEQUENCE_DSA4 AT %IW15390:WORD;
	//Bits comando Alarme Sequence Monitoring Dosador Gravimetrico 5 MECHATRON D-7B linha 1
	STATUS_ALARM_SEQUENCE_DSA5 AT %IW15392: WORD;
	//Bits status Alarme Sequence Monitoring Dosador Gravimetrico 7 MECHATRON D-5A linha 2
	STATUS_ALARM_SEQUENCE_DSA7 AT %IW15394:WORD;
	//Bits status Alarme Sequence Monitoring Dosador Gravimetrico 8 MECHATRON D-7A linha 2	
	STATUS_ALARM_SEQUENCE_DSA8 AT %IW15396:WORD;
	//Bits status Alarme Sequence Monitoring Dosador Gravimetrico 9 MECHATRON D-6A linha 2
	STATUS_ALARM_SEQUENCE_DSA9 AT %IW15398:WORD;
	//Bits status Alarme Sequence Monitoring Dosador Gravimetrico 10 MECHATRON DEA-4A linha 2
	STATUS_ALARM_SEQUENCE_DSA10 AT %IW15400:WORD;
	//Bits status Alarme Sequence Monitoring Dosador Gravimetrico 11 MECHATRON DEA-2A linha 2
	STATUS_ALARM_SEQUENCE_DSA11 AT %IW15402:WORD;
	//Bits status Alarme Sequence Monitoring Dosador Gravimetrico 12 MECHATRON DEA-3A linha 2
	STATUS_ALARM_SEQUENCE_DSA12 AT %IW15404:WORD;
	// Bits status Alarme Sequence Monitoring Dosador Gravimetrico 14
	STATUS_ALARM_SEQUENCE_DSA14 AT %IW15408: WORD;
	//Bits status Alarme Sequence Monitoring Dosador TORRE MECHATRON DEA-D1
	STATUS_ALARM_SEQUENCE_DSATORRE AT %IW15406:WORD;
	
	//Bits status Alarme Maximum Dosador Gravimetrico 1 DEA-600 D-2B linha 1
	STATUS_ALARM_MAXIMUM_DSA1 AT %IW15408:WORD;
	//Bits status Alarme Maximum Dosador Gravimetrico 2 DEA-300 D-4B linha 1
	STATUS_ALARM_MAXIMUM_DSA2 AT %IW15410:WORD;
	//Bits status Alarme Maximum Dosador Gravimetrico 3 DEA-300 D-3B linha 1
	STATUS_ALARM_MAXIMUM_DSA3 AT %IW15412:WORD;
	//Bits status Alarme Maximum Dosador Gravimetrico 4 MECHATRON D-6B linha 1
	STATUS_ALARM_MAXIMUM_DSA4 AT %IW15414:WORD;
	//Bits comando Alarme Maximum Dosador Gravimetrico 5 MECHATRON D-7B linha 1
	STATUS_ALARM_MAXIMUM_DSA5 AT %IW15416:WORD;
	//Bits status Alarme Maximum Dosador Gravimetrico 7 MECHATRON D-5A linha 2
	STATUS_ALARM_MAXIMUM_DSA7 AT %IW15418:WORD;
	//Bits status Alarme Maximum Dosador Gravimetrico 8 MECHATRON D-7A linha 2	
	STATUS_ALARM_MAXIMUM_DSA8 AT %IW15420:WORD;
	//Bits status Alarme Maximum Dosador Gravimetrico 9 MECHATRON D-6A linha 2
	STATUS_ALARM_MAXIMUM_DSA9 AT %IW15422:WORD;
	//Bits status Alarme Maximum Dosador Gravimetrico 10 MECHATRON DEA-4A linha 2
	STATUS_ALARM_MAXIMUM_DSA10 AT %IW15424:WORD;
	//Bits status Alarme Maximum Dosador Gravimetrico 11 MECHATRON DEA-2A linha 2
	STATUS_ALARM_MAXIMUM_DSA11 AT %IW15426:WORD;
	//Bits status Alarme Maximum Dosador Gravimetrico 12 MECHATRON DEA-3A linha 2
	STATUS_ALARM_MAXIMUM_DSA12 AT %IW15428:WORD;
	// Bits status Alarme Maximum Dosador Gravimetrico 14
	STATUS_ALARM_MAXIMUM_DSA14 AT %IW15432: WORD;
	//Bits status Alarme Maximum Dosador TORRE MECHATRON DEA-D1
	STATUS_ALARM_MAXIMUM_DSATORRE AT %IW15430:WORD;
	
	
	//Velocidade em flutuante kg/h Dosador Gravimetrico 1 DEA-600 D-2B linha 1
	PESO_DSA1 AT %QD15060:REAL;	
	//Velocidade em flutuante kg/h Dosador Gravimetrico 2 DEA-300 D-4B linha 1
	PESO_DSA2 AT %QD15064:REAL;
	//Velocidade em flutuante kg/h Dosador Gravimetrico 3 DEA-300 D-3B linha 1	
	PESO_DSA3 AT %QD15068:REAL;
	//Velocidade em flutuante kg/h Dosador Gravimetrico 4 MECHATRON D-6B linha 1
	PESO_DSA4 AT %QD15072:REAL;
	//Velocidade em flutuante kg/h Dosador Gravimetrico 5 MECHATRON D-7B linha 1
	PESO_DSA5 AT %QD15076:REAL;
	//Velocidade em flutuante kg/h Dosador Gravimetrico 7 MECHATRON D-5A linha 2
	PESO_DSA7 AT %QD15080:REAL;
	//Velocidade em flutuante kg/h Dosador Gravimetrico 8 MECHATRON D-7A linha 2	
	PESO_DSA8 AT %QD15084:REAL;
	//Velocidade em flutuante kg/h Dosador Gravimetrico 9 MECHATRON D-6A linha 2
	PESO_DSA9 AT %QD15088:REAL;
	//Velocidade em flutuante kg/h Dosador Gravimetrico 10 MECHATRON DEA-4A linha 2
	PESO_DSA10 AT %QD15092:REAL;
	//Velocidade em flutuante kg/h Dosador Gravimetrico 11 MECHATRON DEA-2A linha 2
	PESO_DSA11 AT %QD15096:REAL;
	//Velocidade em flutuante kg/h Dosador Gravimetrico 12 MECHATRON DEA-3A linha 2
	PESO_DSA12 AT %QD15100:REAL;
	// Velocidade em flutuante kg/h Dosador Gravimetrico 14
	PESO_DSA14 AT %QD15108:REAL;
	//Velocidade em flutuante kg/h Dosador TORRE MECHATRON DEA-D1
	PESO_DSATORRE AT %QD15104:REAL;	
	
	
	
	//Totalizador 1 kg Dosador Gravimetrico 1 DEA-600 D-2B linha 1
	LEITURA_TOTALIZADOR1_DSA1 AT %ID15130:REAL;
	//Totalizador 1 kg Dosador Gravimetrico 2 DEA-300 D-4B linha 1
	LEITURA_TOTALIZADOR1_DSA2 AT %ID15134:REAL;
	//Totalizador 1 kg Dosador Gravimetrico 3 DEA-300 D-3B linha 1
	LEITURA_TOTALIZADOR1_DSA3 AT %ID15138:REAL;
	//Totalizador 1 kg Dosador Gravimetrico 4 MECHATRON D-6B linha 1
	LEITURA_TOTALIZADOR1_DSA4 AT %ID15142:REAL;
	//Totalizador 1 kg Dosador Gravimetrico 5 MECHATRON D-7B linha 1
	LEITURA_TOTALIZADOR1_DSA5 AT %ID15146:REAL;
	//Totalizador 1 kg Dosador Gravimetrico 7 MECHATRON D-5A linha 2
	LEITURA_TOTALIZADOR1_DSA7 AT %ID15150:REAL;
	//Totalizador 1 kg Dosador Gravimetrico 8 MECHATRON D-7A linha 2	
	LEITURA_TOTALIZADOR1_DSA8 AT %ID15154:REAL;
	//Totalizador 1 kg Dosador Gravimetrico 9 MECHATRON D-6A linha 2
	LEITURA_TOTALIZADOR1_DSA9 AT %ID15158:REAL;
	//Totalizador 1 kg Dosador Gravimetrico 10 MECHATRON DEA-4A linha 2
	LEITURA_TOTALIZADOR1_DSA10 AT %ID15162:REAL;
	//Totalizador 1 kg Dosador Gravimetrico 11 MECHATRON DEA-2A linha 2
	LEITURA_TOTALIZADOR1_DSA11 AT %ID15166:REAL;
	//Totalizador 1 kg Dosador Gravimetrico 12 MECHATRON DEA-3A linha 2
	LEITURA_TOTALIZADOR1_DSA12 AT %ID15170:REAL;
	// Totalizador 1 kg Dosador Gravimetrico 14
	LEITURA_TOTALIZADOR1_DSA14 AT %ID15178:REAL;
	//Totalizador 1 kg Dosador TORRE MECHATRON DEA-D1
	LEITURA_TOTALIZADOR1_DSATORRE AT %ID15174:REAL;	
	
	//Totalizador 2 kg Dosador Gravimetrico 1 DEA-600 D-2B linha 1
	LEITURA_TOTALIZADOR2_DSA1 AT %ID15190:REAL;
	//Totalizador 2 kg Dosador Gravimetrico 2 DEA-300 D-4B linha 1
	LEITURA_TOTALIZADOR2_DSA2 AT %ID15194:REAL;
	//Totalizador 2 kg Dosador Gravimetrico 3 DEA-300 D-3B linha 1
	LEITURA_TOTALIZADOR2_DSA3 AT %ID15198:REAL;
	//Totalizador 2 kg Dosador Gravimetrico 4 MECHATRON D-6B linha 1
	LEITURA_TOTALIZADOR2_DSA4 AT %ID15202:REAL;
	//Totalizador 2 kg Dosador Gravimetrico 5 MECHATRON D-7B linha 1
	LEITURA_TOTALIZADOR2_DSA5 AT %ID15206:REAL;
	//Totalizador 2 kg Dosador Gravimetrico 7 MECHATRON D-5A linha 2
	LEITURA_TOTALIZADOR2_DSA7 AT %ID15210:REAL;
	//Totalizador 2 kg Dosador Gravimetrico 8 MECHATRON D-7A linha 2	
	LEITURA_TOTALIZADOR2_DSA8 AT %ID15214:REAL;
	//Totalizador 2 kg Dosador Gravimetrico 9 MECHATRON D-6A linha 2
	LEITURA_TOTALIZADOR2_DSA9 AT %ID15218:REAL;
	//Totalizador 2 kg Dosador Gravimetrico 10 MECHATRON DEA-4A linha 2
	LEITURA_TOTALIZADOR2_DSA10 AT %ID15222:REAL;
	//Totalizador 2 kg Dosador Gravimetrico 11 MECHATRON DEA-2A linha 2
	LEITURA_TOTALIZADOR2_DSA11 AT %ID15226:REAL;
	//Totalizador 2 kg Dosador Gravimetrico 12 MECHATRON DEA-3A linha 2
	LEITURA_TOTALIZADOR2_DSA12 AT %ID15230:REAL;
	// Totalizador 2 kg Dosador Gravimetrico 14
	LEITURA_TOTALIZADOR2_DSA14 AT %ID15238:REAL;
	//Totalizador 2 kg Dosador TORRE MECHATRON DEA-D1
	LEITURA_TOTALIZADOR2_DSATORRE AT %ID15234:REAL;
	
	//Totalizador 3 Ton Dosador Gravimetrico 1 DEA-600 D-2B linha 1
	LEITURA_TOTALIZADOR3_DSA1 AT %ID15300:REAL;
	//Totalizador 3 Ton Dosador Gravimetrico 2 DEA-300 D-4B linha 1
	LEITURA_TOTALIZADOR3_DSA2 AT %ID15304:REAL;
	//Totalizador 3 Ton Dosador Gravimetrico 3 DEA-300 D-3B linha 1
	LEITURA_TOTALIZADOR3_DSA3 AT %ID15308:REAL;
	//Totalizador 3 Ton Dosador Gravimetrico 4 MECHATRON D-6B linha 1
	LEITURA_TOTALIZADOR3_DSA4 AT %ID15312:REAL;
	//Totalizador 3 Ton Dosador Gravimetrico 5 MECHATRON D-7B linha 1
	LEITURA_TOTALIZADOR3_DSA5 AT %ID15316:REAL;
	//Totalizador 3 Ton Dosador Gravimetrico 7 MECHATRON D-5A linha 2
	LEITURA_TOTALIZADOR3_DSA7 AT %ID15320:REAL;
	//Totalizador 3 Ton Dosador Gravimetrico 8 MECHATRON D-7A linha 2	
	LEITURA_TOTALIZADOR3_DSA8 AT %ID15324:REAL;
	//Totalizador 3 Ton Dosador Gravimetrico 9 MECHATRON D-6A linha 2
	LEITURA_TOTALIZADOR3_DSA9 AT %ID15328:REAL;
	//Totalizador 3 Ton Dosador Gravimetrico 10 MECHATRON DEA-4A linha 2
	LEITURA_TOTALIZADOR3_DSA10 AT %ID15332:REAL;
	//Totalizador 3 Ton Dosador Gravimetrico 11 MECHATRON DEA-2A linha 2
	LEITURA_TOTALIZADOR3_DSA11 AT %ID15336:REAL;
	//Totalizador 3 Ton Dosador Gravimetrico 12 MECHATRON DEA-3A linha 2
	LEITURA_TOTALIZADOR3_DSA12 AT %ID15340:REAL;
	// Totalizador 3 Ton Dosador Gravimetrico 14
	LEITURA_TOTALIZADOR3_DSA14 AT %ID15348:REAL;
	//Totalizador 3 Ton Dosador TORRE MECHATRON DEA-D1
	LEITURA_TOTALIZADOR3_DSATORRE AT %ID15344:REAL;

	
	//Leitura Velocidade em flutuante kg/h Dosador Gravimetrico 1 DEA-600 D-2B linha 1
	LEITURA_PESO_DSA1 AT %ID15250:REAL;
	//Leitura Velocidade em flutuante kg/h Dosador Gravimetrico 2 DEA-300 D-4B linha 1
	LEITURA_PESO_DSA2 AT %ID15254:REAL;
	//Leitura Velocidade em flutuante kg/h Dosador Gravimetrico 3 DEA-300 D-3B linha 1
	LEITURA_PESO_DSA3 AT %ID15258:REAL;
	//Leitura Velocidade em flutuante kg/h Dosador Gravimetrico 4 MECHATRON D-6B linha 1
	LEITURA_PESO_DSA4 AT %ID15262:REAL;
	//Leitura Velocidade em flutuante kg/h Dosador Gravimetrico 5 MECHATRON D-7B linha 1
	LEITURA_PESO_DSA5 AT %ID15266:REAL;
	//Leitura Velocidade em flutuante kg/h Dosador Gravimetrico 7 MECHATRON D-5A linha 2
	LEITURA_PESO_DSA7 AT %ID15270:REAL;
	//Leitura Velocidade em flutuante kg/h Dosador Gravimetrico 8 MECHATRON D-7A linha 2	
	LEITURA_PESO_DSA8 AT %ID15274:REAL;
	//Leitura Velocidade em flutuante kg/h Dosador Gravimetrico 9 MECHATRON D-6A linha 2
	LEITURA_PESO_DSA9 AT %ID15278:REAL;
	//Leitura Velocidade em flutuante kg/h Dosador Gravimetrico 10 MECHATRON DEA-4A linha 2
	LEITURA_PESO_DSA10 AT %ID15282:REAL;
	//Leitura Velocidade em flutuante kg/h Dosador Gravimetrico 11 MECHATRON DEA-2A linha 2
	LEITURA_PESO_DSA11 AT %ID15286:REAL;
	//Leitura Velocidade em flutuante kg/h Dosador Gravimetrico 12 MECHATRON DEA-3A linha 2
	LEITURA_PESO_DSA12 AT %ID15290:REAL;
	// Leitura Velocidade em flutuante kg/h Dosador Gravimetrico 14
	LEITURA_PESO_DSA14 AT %ID15298:REAL;
	//Leitura Velocidade em flutuante kg/h Dosador TORRE MECHATRON DEA-D1
	LEITURA_PESO_DSATORRE AT %ID15294:REAL;
	
	//Totalizador 1 realizado inversão Dosador Gravimetrico 1 DEA-600 D-2B linha 1
	TOTALIZADOR1_KG_DS1 AT %QD10000: REAL;
	//Totalizador 2 realizado inversão Dosador Gravimetrico 1 DEA-600 D-2B linha 1
	TOTALIZADOR2_KG_DS1 AT %QD10004: REAL;
	//Totalizador 3 Kg realizado inversão Dosador Gravimetrico 1 DEA-600 D-2B linha 1
	TOTALIZADOR3_KG_DS1 AT %QD10008: REAL;
	//Totalizador 3 TON realizado inversão Dosador Gravimetrico 1 DEA-600 D-2B linha 1	
	TOTALIZADOR3_TON_DS1 AT %QD10012: REAL;
	
	//Totalizador 1 realizado inversão Dosador Gravimetrico 2 DEA-300 D-4B linha 1
	TOTALIZADOR1_KG_DS2 AT %QD10016: REAL;
	//Totalizador 2 realizado inversão Dosador Gravimetrico 2 DEA-300 D-4B linha 1
	TOTALIZADOR2_KG_DS2 AT %QD10020: REAL;
	//Totalizador 3 Kg realizado inversão Dosador Gravimetrico 2 DEA-300 D-4B linha 1
	TOTALIZADOR3_KG_DS2 AT %QD10024: REAL;
	//Totalizador 3 TON realizado inversão Dosador Gravimetrico 2 DEA-300 D-4B linha 1
	TOTALIZADOR3_TON_DS2 AT %QD10028: REAL;
	
	//Totalizador 1 realizado inversão Dosador Gravimetrico 3 DEA-300 D-3B linha 1
	TOTALIZADOR1_KG_DS3 AT %QD10032: REAL;
	//Totalizador 2 realizado inversão Dosador Gravimetrico 3 DEA-300 D-3B linha 1
	TOTALIZADOR2_KG_DS3 AT %QD10036: REAL;
	//Totalizador 3 Kg realizado inversão Dosador Gravimetrico 3 DEA-300 D-3B linha 1
	TOTALIZADOR3_KG_DS3 AT %QD10040: REAL;
	//Totalizador 3 TON realizado inversão Dosador Gravimetrico 3 DEA-300 D-3B linha 1
	TOTALIZADOR3_TON_DS3 AT %QD10044: REAL;
	
	//Totalizador 1 realizado inversão Dosador Gravimetrico 4 MECHATRON D-6B linha 1
	TOTALIZADOR1_KG_DS4 AT %QD10048: REAL;
	//Totalizador 2 realizado inversão Dosador Gravimetrico 4 MECHATRON D-6B linha 1
	TOTALIZADOR2_KG_DS4 AT %QD10052: REAL;
	//Totalizador 3 Kg realizado inversão Dosador Gravimetrico 4 MECHATRON D-6B linha 1
	TOTALIZADOR3_KG_DS4 AT %QD10056: REAL;
	//Totalizador 3 TON realizado inversão Dosador Gravimetrico 4 MECHATRON D-6B linha 1
	TOTALIZADOR3_TON_DS4 AT %QD10060: REAL;
	
	//Totalizador 1 realizado inversão Dosador Gravimetrico 5 MECHATRON D-7B linha 1
	TOTALIZADOR1_KG_DS5 AT %QD10064: REAL;
	//Totalizador 2 realizado inversão Dosador Gravimetrico 5 MECHATRON D-7B linha 1
	TOTALIZADOR2_KG_DS5 AT %QD10068: REAL;
	//Totalizador 3 Kg realizado inversão Dosador Gravimetrico 5 MECHATRON D-7B linha 1
	TOTALIZADOR3_KG_DS5 AT %QD10072: REAL;
	//Totalizador 3 TON realizado inversão Dosador Gravimetrico 5 MECHATRON D-7B linha 1
	TOTALIZADOR3_TON_DS5 AT %QD10076: REAL;
	
	//Totalizador 1 realizado inversão Dosador Gravimetrico 7 MECHATRON D-5A linha 2
	TOTALIZADOR1_KG_DS7 AT %QD10080: REAL;
	//Totalizador 2 realizado inversão Dosador Gravimetrico 7 MECHATRON D-5A linha 2
	TOTALIZADOR2_KG_DS7 AT %QD10084: REAL;
	//Totalizador 3 Kg realizado inversão Dosador Gravimetrico 7 MECHATRON D-5A linha 2
	TOTALIZADOR3_KG_DS7 AT %QD10088: REAL;
	//Totalizador 3 TON realizado inversão Dosador Gravimetrico 7 MECHATRON D-5A linha 2
	TOTALIZADOR3_TON_DS7 AT %QD10092: REAL;
	
	//Totalizador 1 realizado inversão Dosador Gravimetrico 8 MECHATRON D-7A linha 2	
	TOTALIZADOR1_KG_DS8 AT %QD10096: REAL;
	//Totalizador 2 realizado inversão Dosador Gravimetrico 8 MECHATRON D-7A linha 2	
	TOTALIZADOR2_KG_DS8 AT %QD10100: REAL;
	//Totalizador 3 Kg realizado inversão Dosador Gravimetrico 8 MECHATRON D-7A linha 2	
	TOTALIZADOR3_KG_DS8 AT %QD10104: REAL;
	//Totalizador 3 TON realizado inversão Dosador Gravimetrico 8 MECHATRON D-7A linha 2	
	TOTALIZADOR3_TON_DS8 AT %QD10108: REAL;
	
	//Totalizador 1 realizado inversão Dosador Gravimetrico 9 MECHATRON D-6A linha 2	
	TOTALIZADOR1_KG_DS9 AT %QD10112: REAL;
	//Totalizador 2 realizado inversão Dosador Gravimetrico 9 MECHATRON D-6A linha 2	
	TOTALIZADOR2_KG_DS9 AT %QD10116: REAL;
	//Totalizador 3 Kg realizado inversão Dosador Gravimetrico 9 MECHATRON D-6A linha 2
	TOTALIZADOR3_KG_DS9 AT %QD10120: REAL;
	//Totalizador 3 TON realizado inversão Dosador Gravimetrico 9 MECHATRON D-6A linha 2	
	TOTALIZADOR3_TON_DS9 AT %QD10124: REAL;
	
	//Totalizador 1 realizado inversão Dosador Gravimetrico 10 MECHATRON DEA-4A linha 2	
	TOTALIZADOR1_KG_DS10 AT %QD10128: REAL;
	//Totalizador 2 realizado inversão Dosador Gravimetrico 10 MECHATRON DEA-4A linha 2	
	TOTALIZADOR2_KG_DS10 AT %QD10132: REAL;
	//Totalizador 3 Kg realizado inversão Dosador Gravimetrico 10 MECHATRON DEA-4A linha 2
	TOTALIZADOR3_KG_DS10 AT %QD10136: REAL;
	//Totalizador 3 TON realizado inversão Dosador Gravimetrico 10 MECHATRON DEA-4A linha 2	
	TOTALIZADOR3_TON_DS10 AT %QD10140: REAL;
	
	//Totalizador 1 realizado inversão Dosador Gravimetrico 11 MECHATRON DEA-2A linha 2	
	TOTALIZADOR1_KG_DS11 AT %QD10144: REAL;
	//Totalizador 2 realizado inversão Dosador Gravimetrico 11 MECHATRON DEA-2A linha 2	
	TOTALIZADOR2_KG_DS11 AT %QD10148: REAL;
	//Totalizador 3 Kg realizado inversão Dosador Gravimetrico 11 MECHATRON DEA-2A linha 2
	TOTALIZADOR3_KG_DS11 AT %QD10152: REAL;
	//Totalizador 3 TON realizado inversão Dosador Gravimetrico 11 MECHATRON DEA-2A linha 2
	TOTALIZADOR3_TON_DS11 AT %QD10156: REAL;
	
	//Totalizador 1 realizado inversão Dosador Gravimetrico 12 MECHATRON DEA-3A linha 2	
	TOTALIZADOR1_KG_DS12 AT %QD10160: REAL;
	//Totalizador 2 realizado inversão Dosador Gravimetrico 12 MECHATRON DEA-3A linha 2
	TOTALIZADOR2_KG_DS12 AT %QD10164: REAL;
	//Totalizador 3 Kg realizado inversão Dosador Gravimetrico 12 MECHATRON DEA-3A linha 2
	TOTALIZADOR3_KG_DS12 AT %QD10168: REAL;
	//Totalizador 3 TON realizado inversão Dosador Gravimetrico 12 MECHATRON DEA-3A linha 2
	TOTALIZADOR3_TON_DS12 AT %QD10172: REAL;
	
	// Totalizador 1 realizado inversão Dosador Gravimetrico 14
	TOTALIZADOR1_KG_DS14 AT %QD20160: REAL;
	// Totalizador 2 realizado inversão Dosador Gravimetrico 14
	TOTALIZADOR2_KG_DS14 AT %QD20164: REAL;
	// Totalizador 3 Kg realizado inversão Dosador Gravimetrico 14
	TOTALIZADOR3_KG_DS14 AT %QD20168: REAL;
	// Totalizador 3 TON realizado inversão Dosador Gravimetrico 14
	TOTALIZADOR3_TON_DS14 AT %QD20172: REAL;
	
	//Totalizador 1 realizado inversão Dosador TORRE MECHATRON DEA-D1	
	TOTALIZADOR1_KG_DSTORRE AT %QD10176: REAL;
	//Totalizador 2 realizado inversão Dosador TORRE MECHATRON DEA-D1
	TOTALIZADOR2_KG_DSTORRE AT %QD10180: REAL;
	//Totalizador 3 Kg realizado inversão Dosador TORRE MECHATRON DEA-D1
	TOTALIZADOR3_KG_DSTORRE AT %QD10184: REAL;
	//Totalizador 3 TON realizado inversão Dosador TORRE MECHATRON DEA-D1
	TOTALIZADOR3_TON_DSTORRE AT %QD10188: REAL;
	
	//Velocidade real do Dosador Gravimetrico 1 DEA-600 D-2B linha 1
	VELOCIDADE_REAL_DS1 AT %QD10192:REAL;
	//Velocidade real do Dosador Gravimetrico 2 DEA-300 D-4B linha 1
	VELOCIDADE_REAL_DS2 AT %QD10196:REAL;
	//Velocidade real do Dosador Gravimetrico 3 DEA-300 D-3B linha 1
	VELOCIDADE_REAL_DS3 AT %QD10200:REAL;
	//Velocidade real do Dosador Gravimetrico 4 MECHATRON D-6B linha 1
	VELOCIDADE_REAL_DS4 AT %QD10204:REAL;
	//Velocidade real do Dosador Gravimetrico 5 MECHATRON D-7B linha 1
	VELOCIDADE_REAL_DS5 AT %QD10208:REAL;		
	//Velocidade real do Dosador Gravimetrico 7 MECHATRON D-5A linha 2
	VELOCIDADE_REAL_DS7 AT %QD10212:REAL;
	//Velocidade real do Dosador Gravimetrico 8 MECHATRON D-7A linha 2
	VELOCIDADE_REAL_DS8 AT %QD10216:REAL;
	//Velocidade real do Dosador Gravimetrico 9 MECHATRON D-6A linha 2
	VELOCIDADE_REAL_DS9 AT %QD10220:REAL;
	//Velocidade real do Dosador Gravimetrico 10 MECHATRON DEA-4A linha 2	
	VELOCIDADE_REAL_DS10 AT %QD10224: REAL;
	//Velocidade real do Dosador Gravimetrico 11 MECHATRON DEA-2A linha 2
	VELOCIDADE_REAL_DS11 AT %QD10228: REAL;
	//Velocidade real do Dosador Gravimetrico 12 MECHATRON DEA-3A linha 2
	VELOCIDADE_REAL_DS12 AT %QD10232:REAL;
	// Velocidade real do Dosador Gravimetrico 14
	VELOCIDADE_REAL_DS14 AT %QD20232:REAL;
	//Velocidade real do Dosador TORRE MECHATRON DEA-D1
	VELOCIDADE_REAL_DSTORRE AT %QD10236:REAL;

	//Velocidade real do Dosador 1
	VELOCIDADE_REAL2_DS1 AT %QD10300:REAL;
	//Velocidade real do Dosador 2
	VELOCIDADE_REAL2_DS2 AT %QD10304:REAL;
	//Velocidade real do Dosador 3
	VELOCIDADE_REAL2_DS3 AT %QD10308:REAL;
	//Velocidade real do Dosador 4
	VELOCIDADE_REAL2_DS4 AT %QD10312:REAL;
	//Velocidade real do Dosador 5
	VELOCIDADE_REAL2_DS5 AT %QD10316:REAL;
	//Velocidade real do Dosador 7
	VELOCIDADE_REAL2_DS7 AT %QD10320:REAL;
	//Velocidade real do Dosador 8
	VELOCIDADE_REAL2_DS8 AT %QD10324:REAL;
	//Velocidade real do Dosador 9
	VELOCIDADE_REAL2_DS9 AT %QD10328:REAL;
	//Velocidade real do Dosador 10
	VELOCIDADE_REAL2_DS10 AT %QD10332:REAL;
	//Velocidade real do Dosador 11
	VELOCIDADE_REAL2_DS11 AT %QD10336:REAL;
	//Velocidade real do Dosador 12
	VELOCIDADE_REAL2_DS12 AT %QD10340:REAL;
	// Velocidade real do Dosador 14
	VELOCIDADE_REAL2_DS14 AT %QD10548:REAL;
	//Velocidade real do Dosador Torre
	VELOCIDADE_REAL2_DSTORRE AT %QD10344:REAL;
	
			
			

	
	
END_VAR

// Supervisório
VAR_GLOBAL PERSISTENT
	
	//Botão comando modo volumetrico - dosador Gravimetrico 1 DEA-600 D-2B linha 1		
	BTS_MODVOL_DS1 AT %QX3010.1:BOOL;	
	//Botão comando modo gravimetrico - dosador Gravimetrico 1 DEA-600 D-2B linha 1	
	BTS_MODGRAV_DS1 AT %QX3010.2:BOOL;
	//Botão comando modo volumetrico - dosador Gravimetrico 2 DEA-300 D-4B linha 1		 
	BTS_MODVOL_DS2 AT %QX3010.6:BOOL;		
	//Botão comando modo gravimetrica - dosador Gravimetrico 2 DEA-300 D-4B linha 1	
	BTS_MODGRAV_DS2 AT %QX3010.7:BOOL;
	//Botão comando modo volumetrico - dosador Gravimetrico 3 DEA-300 D-3B linha 1	
	BTS_MODVOL_DS3 AT %QX3011.3:BOOL;		
	//Botão comando modo gravimetrica - dosador Gravimetrico 3 DEA-300 D-3B linha 1	
	BTS_MODGRAV_DS3 AT %QX3011.4:BOOL;
	//Botão comando modo volumetrico - dosador Gravimetrico 4 MECHATRON D-6B linha 1	
	BTS_MODVOL_DS4 AT %QX3012.0:BOOL;		
	//Botão comando modo graviemtrico - dosador Gravimetrico 4 MECHATRON D-6B linha 1	
	BTS_MODGRAV_DS4 AT %QX3012.1:BOOL;	
	//Botão comando modo volumetrico - dosador Gravimetrico 5 MECHATRON D-7B linha 1	
	BTS_MODVOL_DS5 AT %QX3012.5	:BOOL;	
	//Botão comando modo graviemtrico - dosador Gravimetrico 5 MECHATRON D-7B linha 1	
	BTS_MODGRAV_DS5 AT %QX3012.6:BOOL;	
	//Botão comando modo volumetrico - dosador Gravimetrico 7 MECHATRON D-5A linha 2
	BTS_MODVOL_DS7 AT %QX3013.2:BOOL;		
	//Botão comando modo gravimetrico - dosador Gravimetrico 7 MECHATRON D-5A linha 2
	BTS_MODGRAV_DS7 AT %QX3013.3:BOOL;	
	//Botão comando modo volumetrico - dosador Gravimetrico 8 MECHATRON D-7A linha 2
	BTS_MODVOL_DS8 AT %QX3013.7:BOOL;
	//Botão comando modo gravimetrico - dosador Gravimetrico 8 MECHATRON D-7A linha 2
	BTS_MODGRAV_DS8 AT %QX3014.0:BOOL;
	//Botão comando modo volumetrico - dosador Gravimetrico 9 MECHATRON D-6A linha 2
	BTS_MODVOL_DS9 AT %QX3014.4:BOOL;
	//Botão comando modo graviemtrico - dosador Gravimetrico 9 MECHATRON D-6A linha 2
	BTS_MODGRAV_DS9 AT %QX3014.5:BOOL;	
	//Botão comando modo volumetrico - dosador Gravimetrico 10 MECHATRON DEA-4A linha 2
	BTS_MODVOL_DS10 AT %QX3015.1:BOOL;
	//Botão comando modo graviemtrico - dosador Gravimetrico 10 MECHATRON DEA-4A linha 2
	BTS_MODGRAV_DS10 AT %QX3015.2:BOOL;
	//Botão comando modo volumetrico - dosador Gravimetrico 11 MECHATRON DEA-2A linha 2
	BTS_MODVOL_DS11 AT %QX3015.6:BOOL;
	//Botão comando modo gravimetrico - dosado Gravimetrico 11 MECHATRON DEA-2A linha 2
	BTS_MODGRAV_DS11 AT %QX3015.7:BOOL;
	//Botão comando modo volumetrico - dosador Gravimetrico 12 MECHATRON DEA-3A linha 2
	BTS_MODVOL_DS12 AT %QX3016.3:BOOL;
	//Botão comando modo gravimetrico - dosador Gravimetrico 12 MECHATRON DEA-3A linha 2
	BTS_MODGRAV_DS12 AT %QX3016.4:BOOL;
	// Botão comando modo volumetrico - dosador Gravimetrico 14
	BTS_MODVOL_DS14 AT %QX3022.1:BOOL;
	// Botão comando modo gravimetrico - dosador Gravimetrico 14
	BTS_MODGRAV_DS14 AT %QX3022.3:BOOL;
	//Botão comando modo volumetrico - dosador Sulfato torre  MECHATRON DEA-D1
	BTS_MODVOL_DSTORRE AT %QX3017.0:BOOL;
	//Botão comando modo gravimetrico - dosador Sulfato torre  MECHATRON DEA-D1
	BTS_MODGRAV_DSTORRE AT %QX3017.1:BOOL;			


END_VAR

// Device/Application/IOQualities
VAR_GLOBAL
	QUALITY_NX1001: ARRAY[0..15] OF LibDataTypes.QUALITY;
	QUALITY_NX1001_01: ARRAY[0..15] OF LibDataTypes.QUALITY;
	QUALITY_NX1001_02: ARRAY[0..15] OF LibDataTypes.QUALITY;
	QUALITY_NX1001_03: ARRAY[0..15] OF LibDataTypes.QUALITY;
	QUALITY_NX1001_04: ARRAY[0..15] OF LibDataTypes.QUALITY;
	QUALITY_NX1001_05: ARRAY[0..15] OF LibDataTypes.QUALITY;
	QUALITY_NX1001_06: ARRAY[0..15] OF LibDataTypes.QUALITY;
	QUALITY_NX2001: ARRAY[0..15] OF LibDataTypes.QUALITY;
	QUALITY_NX2001_01: ARRAY[0..15] OF LibDataTypes.QUALITY;
	QUALITY_NX2001_02: ARRAY[0..15] OF LibDataTypes.QUALITY;
	QUALITY_NX2001_03: ARRAY[0..15] OF LibDataTypes.QUALITY;
	QUALITY_NX2001_04: ARRAY[0..15] OF LibDataTypes.QUALITY;
	QUALITY_NX2001_05: ARRAY[0..15] OF LibDataTypes.QUALITY;
	QUALITY_NX2001_06: ARRAY[0..15] OF LibDataTypes.QUALITY;
	QUALITY_NX6000: ARRAY[0..7] OF LibDataTypes.QUALITY;
	QUALITY_NX6000_01: ARRAY[0..7] OF LibDataTypes.QUALITY;
	QUALITY_NX6000_02: ARRAY[0..7] OF LibDataTypes.QUALITY;
	QUALITY_NX6000_03: ARRAY[0..7] OF LibDataTypes.QUALITY;
	QUALITY_NX6010: ARRAY[0..7] OF LibDataTypes.QUALITY;
	QUALITY_NX6100: ARRAY[0..3] OF LibDataTypes.QUALITY;
	QUALITY_NX6100_01: ARRAY[0..3] OF LibDataTypes.QUALITY;
	QUALITY_NX6100_02: ARRAY[0..3] OF LibDataTypes.QUALITY;
END_VAR

// Device/Application/Special_Variables
(*This GVL is blocked to edit.*)
VAR_GLOBAL
	Pulse_100ms : BOOL;                     //Pulse signal with 100ms period (toggles every 50ms)
	Pulse_500ms : BOOL;                     //Pulse signal with 500ms period (toggles every 250ms)
	Pulse_1s    : BOOL;                     //Pulse signal with 1s period (toggles every 500ms)
	Pulse_2s    : BOOL;                     //Pulse signal with 2s period (toggles every 1s)
	Pulse_5s    : BOOL;                     //Pulse signal with 5s period (toggles every 2,5s)
	Pulse_10s   : BOOL;                     //Pulse signal with 10s period (toggles every 5s)
	Pulse_30s   : BOOL;                     //Pulse signal with 30s period (toggles every 15s)
	Pulse_60s   : BOOL;                     //Pulse signal with 60s period (toggles every 30s)
	Pulse_Scan  : BOOL;                     //Scan pulse that toggles every MainTask cycle
	System_Time : EXTENDED_DATE_AND_TIME;   //System date and time
	Day_Of_Week : DAYS_OF_WEEK;             //Day of week
	Hour_Minute : UINT;                     //Integer variable with hour and minute (hour*100 + minute)
END_VAR

VAR_GLOBAL CONSTANT
	udiMainTaskInterval : UDINT := 100000;     //MainTask configured interval [us].
END_VAR

// Device/Application/GVL_Ampliacao_transferencia



VAR_GLOBAL
	// status motor moinho 01
	MH_01_STS AT %QX15112.0: BOOL;
	// comando liga moinho 01
	MH_01_CMDS AT %QX15122.3: BOOL;
	// falha inversor do moinho 01
	MH_01_FLTS AT %QX15112.1: BOOL;
	// status motor moinho 02 sup
	MH_02_STS AT %QX15112.2: BOOL;
	// comando liga moinho 02 sup
	MH_02_CMDS AT %QX15122.0: BOOL;
	// falha inversor do moinho 02 sup
	MH_02_FLTS AT %QX15112.3: BOOL;
	// status motor bomba de baixa 02 sup
	BB_02_STS AT %QX15112.4: BOOL;
	// comando liga bomba de baixa 02 sup
	BB_02_CMDS AT %QX15122.1: BOOL;
	// falha inversor bomba de baixa 02 sup
	BB_02_FLTS AT %QX15112.5: BOOL;
	// status motor bomba de alta 03 sup
	BA_03_STS AT %QX15112.6: BOOL;
	// comando liga bomba de alta 03 sup
	BA_03_CMDS AT %QX15122.2: BOOL;
	// falha inversor bomba de alta 03 sup
	BA_03_FLTS AT %QX15112.7: BOOL;
	// falha motor bomba lubrificação 03 sup
	BL_03_FLTS AT %QX15120.0: BOOL;
	// preset velocidade da bomba de baixa 02  sup
	BB_02_PST_VELS AT %QW15114: WORD;
	// velocidade da bomba de alta 03 sup
	BA_03_ST_VELS AT %QW15116: WORD;
	// pressotato da bomba de baixa 02 sup
	BB_02_PRTS AT %QW15118: WORD;
	// status leitura do inversor bomba alta 03
	BA_03_INV_LEITURA AT %QW1600: DWORD;
	// status escrita do inversor bomba alta 03
	BA_03_INV_ESCRITA AT %IW1600: DWORD;
	// status leitura do inversor bomba baixa 02
	BB_02_INV_LEITURA AT %QW1604: DWORD;
	// status escrita do inversor bomba baixa 02
	BB_02_INV_ESCRITA AT %IW1604: DWORD;
	// status leitura do inversor moinho 01
	MH_01_INV_LEITURA AT %QW1608: DWORD;
	// status escrita do inversor moinho 01
	MH_01_INV_ESCRITA AT %IW1608: DWORD;
	// status leitura do inversor moinho 02
	MH_02_INV_LEITURA AT %QW1612: DWORD;
	// status escrita do inversor moinho 02
	MH_02_INV_ESCRITA AT %IW1612: DWORD;
	// comando liga inversor bomba alta 03
	BA_03_CMD AT %IX1600.0: BOOL;
	// comando habilita inversor bomba alta 03
	BA_03_HAB AT %IX1600.1: BOOL;
	// parada de emergencia inversor bomba de alta 03
	BA_03_STP AT %IX1600.6: BOOL;
	// reset de falha inversor bomba de alta 03
	BA_03_RST AT %IX1600.7: BOOL;
	// status do inversor da bomba de alta 03
	BA_03_ST AT %QX1601.1: BOOL;
	// indicação de falha do inversor da bomba de alta 03
	BA_03_FLT AT %QX1601.7: BOOL;
	// comando liga inversor bomba baixa 02
	BB_02_CMD AT %IX1604.0: BOOL;
	// comando habilita inversor bomba baixa 02
	BB_02_HAB AT %IX1604.1: BOOL;
	// parada de emergencia inversor bomba de baixa 02
	BB_02_STP AT %IX1604.6: BOOL;
	// reset de falha inversor bomba de baixa 02
	BB_02_RST AT %IX1604.7: BOOL;
	// status do inversor da bomba de baixa 02
	BB_02_ST AT %QX1605.1: BOOL;
	// indicação de falha do inversor da bomba de baixa 02
	BB_02_FLT AT %QX1605.7: BOOL;
	// comando liga inversor moinho 01
	MH_01_CMD AT %IX1608.0: BOOL;
	// comando habilita inversor moinho 01
	MH_01_HAB AT %IX1608.1: BOOL;
	// parada de emergencia inversor moinho 01
	MH_01_STP AT %IX1608.6: BOOL;
	// reset de falha inversor moinho 01
	MH_01_RST AT %IX1608.7: BOOL;
	// status do inversor moinho 01
	MH_01_ST AT %QX1609.1: BOOL;
	// indicação de falha do inversor moinho 01
	MH_01_FLT AT %QX1609.7: BOOL;
	// comando liga inversor moinho 02
	MH_02_CMD AT %IX1612.0: BOOL;
	// comando habilita inversor moinho 02
	MH_02_HAB AT %IX1612.1: BOOL;
	// parada de emergencia inversor moinho 02
	MH_02_STP AT %IX1612.6: BOOL;
	// reset de falha inversor moinho 02
	MH_02_RST AT %IX1612.7: BOOL;
	// status do inversor moinho 02
	MH_02_ST AT %QX1613.1: BOOL;
	// indicação de falha do inversor moinho 02
	MH_02_FLT AT %QX1613.7: BOOL;
	// referencia de velocidade do inversor da bomba de alta 03
	BA_03_PRS_VEL AT %IW1602: WORD;
	// velocidade atual do inversor da bomba de alta 03
	BA_03_REF_VEL AT %QW1602: WORD;
	// referencia de velocidade do inversor da bomba de baixa 02
	BB_02_PRS_VEL AT %IW1606: WORD;
	// velocidade atual do inversor da bomba de baixa 02
	BB_02_REF_VEL AT %QW1606: WORD;
	PRESSAO_BOMBA AT %MW1600: REAL;
	// falha do pressostato da bomba de alta 03
	BA_03_FLT_PRESS AT %QX15113.0: BOOL;
	
	
END_VAR

// Device/Application/MainPrg
PROGRAM MainPrg
VAR
END_VAR

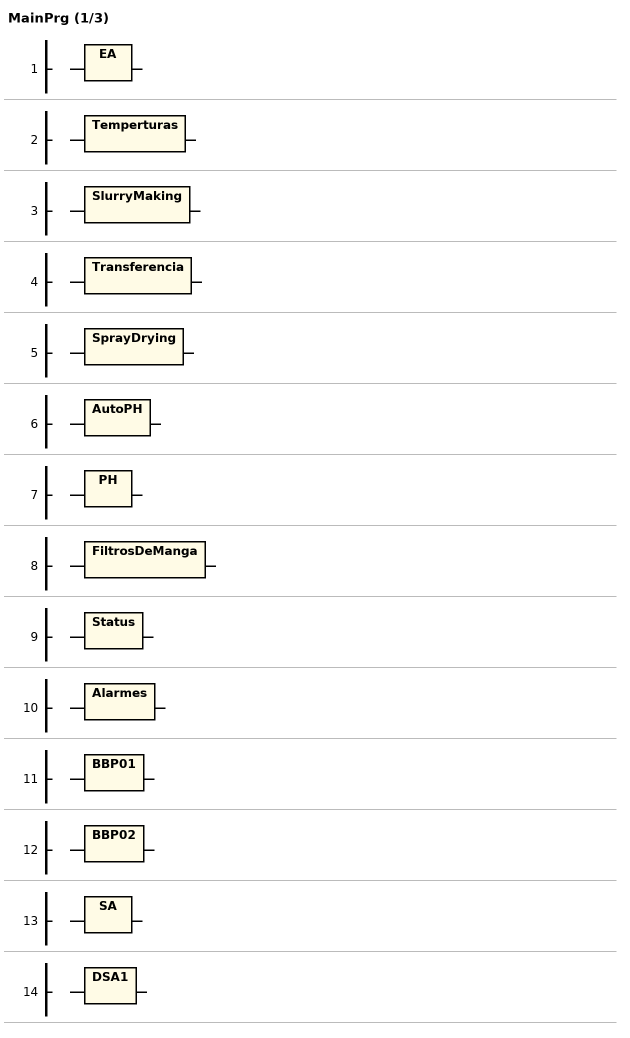
// NETWORK 1
EA();

// NETWORK 2
Temperturas();

// NETWORK 3
SlurryMaking();

// NETWORK 4
Transferencia();

// NETWORK 5
SprayDrying();

// NETWORK 6
AutoPH();

// NETWORK 7
PH();

// NETWORK 8
FiltrosDeManga();

// NETWORK 9
Status();

// NETWORK 10
Alarmes();

// NETWORK 11
BBP01();

// NETWORK 12
BBP02();

// NETWORK 13
SA();

// NETWORK 14
DSA1();

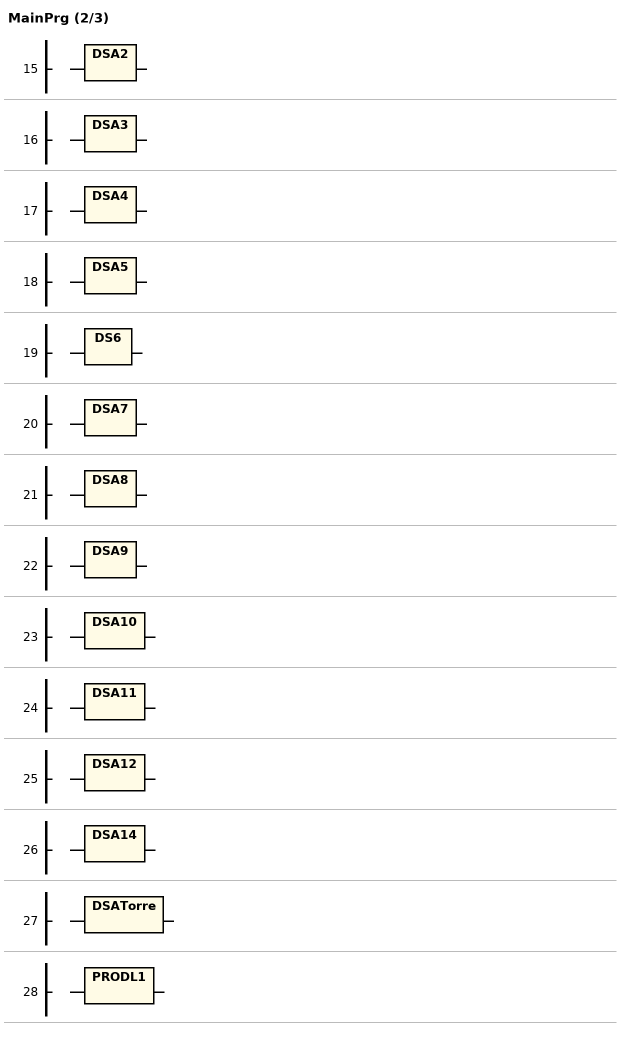
// NETWORK 15
DSA2();

// NETWORK 16
DSA3();

// NETWORK 17
DSA4();

// NETWORK 18
DSA5();

// NETWORK 19
DS6();

// NETWORK 20
DSA7();

// NETWORK 21
DSA8();

// NETWORK 22
DSA9();

// NETWORK 23
DSA10();

// NETWORK 24
DSA11();

// NETWORK 25
DSA12();

// NETWORK 26
DSA14();

// NETWORK 27
DSATorre();

// NETWORK 28
PRODL1();

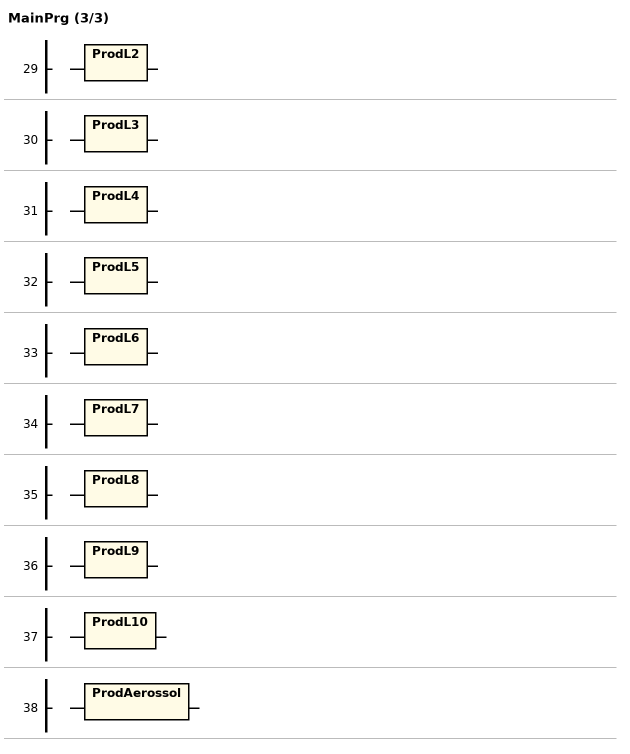
// NETWORK 29
ProdL2();

// NETWORK 30
ProdL3();

// NETWORK 31
ProdL4();

// NETWORK 32
ProdL5();

// NETWORK 33
ProdL6();

// NETWORK 34
ProdL7();

// NETWORK 35
ProdL8();

// NETWORK 36
ProdL9();

// NETWORK 37
ProdL10();

// NETWORK 38
ProdAerossol();

END_PROGRAM

// Device/Application/EA
PROGRAM EA
VAR
	
	//converte escala entrada analogica 1 (peso balança solidos 1)
	converteEA1:LIN_TRAFO;
	//converte escala entrada analogica 2 (peso balança solidos 2)
	converteEA2:LIN_TRAFO;
	//converte escala entrada analogica 3 (peso balança solidos 3)
	converteEA3:LIN_TRAFO;
	//converte escala entrada analogica 4 (peso balança solidos 4)
	converteEA4:LIN_TRAFO;
	//converte escala entrada analogica 5 (peso balança solidos 5)
	converteEA5:LIN_TRAFO;
	//converte escala entrada analogica 6 (peso balança liquidos 1)
	converteEA6:LIN_TRAFO;
	//converte escala entrada analogica 7 (peso balança liquidos 2)
	converteEA7:LIN_TRAFO;
	//converte escala entrada analogica 8 (peso balança liquidos 3)
	converteEA8:LIN_TRAFO;
	//converte escala entrada analogica 1 01 (peso balança liquidos 4)
	converteEA101:LIN_TRAFO;
	//converte escala entrada analogica 2 01 (pressão linha de alta)
	converteEA201:LIN_TRAFO;
	//converte escala entrada analogica 3 01 (pressão linha de baixa)
	converteEA301:LIN_TRAFO;
	//converte escala entrada analogica 4 01 (Nivel misturador principal)
	converteEA401:LIN_TRAFO;
	//converte escala entrada analogica 5 01 (Nivel mexedor de espera principal)
	converteEA501:LIN_TRAFO;
	//converte escala entrada analogica 6 01 (Velocidade bomba alta 1)
	converteEA601:LIN_TRAFO;
	//converte escala entrada analogica 7 01 (Velocidade bomba alta 2)
	converteEA701:LIN_TRAFO;
	//converte escala entrada analogica 8 01 (Pressao da torre bomba alta 2)
	converteEA801:LIN_TRAFO;
	//converte escala entrada analogica 1 02 (Peso do fluidizador 1)
	converteEA102:LIN_TRAFO;
	//converte escala entrada analogica 2 02 (Peso do fluidizador 2)
	converteEA202:LIN_TRAFO;
	// converte escala entrada analogica 502 (Fluxo BBP02)
	converteEA502: LIN_TRAFO;
	// converte escala entrada analogica 502 (Fluxo BBP01)
	converteEA702: LIN_TRAFO;
	// converte escala entrada analogica 402 (umidade)
	converteEA402: LIN_TRAFO;
	// Medição de umidade infrared
	//VALOR_MEDICAO_UMIDADE: REAL;
	// converte escala entrada analogica 302 (temperatura torre)
	converteEA302: LIN_TRAFO;
	BLINK_0: BLINK;
	HABIL_ATUAL_FLUI1: BOOL;
	LEITURA_PESO_FLUI1_INST: REAL;
	BLINK_1: BLINK;
	HABIL_ATUAL_FLUI2: BOOL;
	LEITURA_PESO_FLUI2_INST: REAL;
	converteEA602: LIN_TRAFO;
	OUT: INT;
	converteEA303: LIN_TRAFO;
	// Sensor de temperatura na tubulação entrada da torre
	converteEA103: LIN_TRAFO;
	// Sensor de temperatura na tubulação de liberação para atmosfera
	converteEA203: LIN_TRAFO;
	converteEA403: LIN_TRAFO;
END_VAR

VAR_INPUT
	IN: INT;
	IN_MIN: INT;
	IN_MAX: INT;
	OUT_MIN: INT;
	OUT_MAX: INT;
END_VAR

// ===========================================================================================
// POU de conversão das entradas analógicas
//============================================================================================


// Entrada analógica 1 : NX6000 - Peso da Balanca de Solido 1  ( kg mA) ===================================================== 
converteEA1(IN:=EA1, IN_MIN:=PRST_INI_ESCA_ENG_BLS1, IN_MAX:=PRST_FIM_ESCA_ENG_BLS1,OUT_MIN:=0, OUT_MAX:=PRST_FIM_ESCA_KG_BLS1);
LEITURA_PESO_BLS1:= converteEA1.OUT;
LEITURA_REAL_ENGE_BLS1 := INT_TO_REAL(EA1);

// Entrada analógica 2 : NX6000 - Peso da Balanca de Solido 2  ( kg mA) ===================================================== 
converteEA2(IN:=EA2, IN_MIN:=PRST_INI_ESCA_ENG_BLS2, IN_MAX:=PRST_FIM_ESCA_ENG_BLS2,OUT_MIN:=0, OUT_MAX:=PRST_FIM_ESCA_KG_BLS2);
LEITURA_PESO_BLS2:= converteEA2.OUT;
LEITURA_REAL_ENGE_BLS2 := INT_TO_REAL(EA2);

// Entrada analógica 3 : NX6000 - Peso da Balanca de Solido 3  ( kg mA) ===================================================== 
converteEA3(IN:=EA3, IN_MIN:=PRST_INI_ESCA_ENG_BLS3, IN_MAX:=PRST_FIM_ESCA_ENG_BLS3,OUT_MIN:=0, OUT_MAX:=PRST_FIM_ESCA_KG_BLS3);
LEITURA_PESO_BLS3:= converteEA3.OUT;
LEITURA_REAL_ENGE_BLS3 := INT_TO_REAL(EA3);

// Entrada analógica 4 : NX6000 - Peso da Balanca de Solido 4  ( kg mA) ===================================================== 
converteEA4(IN:=EA4, IN_MIN:=PRST_INI_ESCA_ENG_BLS4, IN_MAX:=PRST_FIM_ESCA_ENG_BLS4,OUT_MIN:=0, OUT_MAX:=PRST_FIM_ESCA_KG_BLS4);
LEITURA_PESO_BLS4:= converteEA4.OUT;
LEITURA_REAL_ENGE_BLS4 := INT_TO_REAL(EA4);

// Entrada analógica 5 : NX6000 - Peso da Balanca de Solido 5  ( kg mA) ===================================================== 
converteEA5(IN:=EA5, IN_MIN:=PRST_INI_ESCA_ENG_BLS5, IN_MAX:=PRST_FIM_ESCA_ENG_BLS5,OUT_MIN:=0, OUT_MAX:=PRST_FIM_ESCA_KG_BLS5);
LEITURA_PESO_BLS5:= converteEA5.OUT;
LEITURA_REAL_ENGE_BLS5 := INT_TO_REAL(EA5);

// Entrada analógica 6 : NX6000 - Peso da Balanca de Liquidos 1  ( kg mA) ===================================================== 
converteEA6(IN:=EA6, IN_MIN:=PRST_INI_ESCA_ENG_BLL1, IN_MAX:=PRST_FIM_ESCA_ENG_BLL1,OUT_MIN:=0, OUT_MAX:=PRST_FIM_ESCA_KG_BLL1);
LEITURA_PESO_BLL1:= converteEA6.OUT;
LEITURA_REAL_ENGE_BLL1 := INT_TO_REAL(EA6);

// Entrada analógica 7 : NX6000 - Peso da Balanca de Liquidos 2  ( kg mA) ===================================================== 
converteEA7(IN:=EA7, IN_MIN:=PRST_INI_ESCA_ENG_BLL2, IN_MAX:=PRST_FIM_ESCA_ENG_BLL2,OUT_MIN:=0, OUT_MAX:=PRST_FIM_ESCA_KG_BLL2);
LEITURA_PESO_BLL2:= converteEA7.OUT;
LEITURA_REAL_ENGE_BLL2 := INT_TO_REAL(EA7);

// Entrada analógica 8 : NX6000 - Peso da Balanca de Liquidos 3  ( kg mA) ===================================================== 
converteEA8(IN:=EA8, IN_MIN:=PRST_INI_ESCA_ENG_BLL3, IN_MAX:=PRST_FIM_ESCA_ENG_BLL3,OUT_MIN:=0, OUT_MAX:=PRST_FIM_ESCA_KG_BLL3);
LEITURA_PESO_BLL3:= converteEA8.OUT;
LEITURA_REAL_ENGE_BLL3 := INT_TO_REAL(EA8);

// Entrada analógica 1 : NX6000_1 - Peso da Balanca de Liquidos 4  ( kg mA) ===================================================== 
converteEA101(IN:=EA101, IN_MIN:=PRST_INI_ESCA_ENG_BLL4, IN_MAX:=PRST_FIM_ESCA_ENG_BLL4,OUT_MIN:=0, OUT_MAX:=PRST_FIM_ESCA_KG_BLL4);
LEITURA_PESO_BLL4:= converteEA101.OUT;
LEITURA_REAL_ENGE_BLL4 := INT_TO_REAL(EA101);

// Entrada analógica 2 : NX6000_1 - Pressão linha de alta ( bar mA) ===================================================== 
converteEA201(IN:=EA201, IN_MIN:=0, IN_MAX:=4000,OUT_MIN:=0, OUT_MAX:=70);
LEITURA_PRES_LA:= converteEA201.OUT;


// Entrada analógica 3 : NX6000_1 - Pressão linha de baixa ( bar mA) ===================================================== 
converteEA301(IN:=EA301, IN_MIN:=0, IN_MAX:=3000,OUT_MIN:=0, OUT_MAX:=12);
LEITURA_PRES_LB:= converteEA301.OUT;


// Entrada analógica 4 : NX6000_1 - Peso misturador principal ( 0-6000Kg mA) ===================================================== 
converteEA401(IN:=EA401, IN_MIN:=0, IN_MAX:=4000,OUT_MIN:=0, OUT_MAX:=6000);
//se o valor for menor que minimo, zera
IF EA401<5 THEN
	LEITURA_NI_MISTPRIN:=0;
ELSE
	LEITURA_NI_MISTPRIN:= converteEA401.OUT;
END_IF


// Entrada analógica 5 : NX6000_1 - Nivel mexedor de espera ( 0-100.0% mA) ===================================================== 
converteEA501(IN:=EA501, IN_MIN:=5, IN_MAX:=3100,OUT_MIN:=0, OUT_MAX:=100);
//se o valor for menor que minimo, zera
IF EA501<5 THEN
	LEITURA_NI_MXESPE:= 0;
ELSE
	LEITURA_NI_MXESPE:= converteEA501.OUT;
END_IF


// Entrada analógica 6 : NX6000_1 - Leitura velocidade bomba alta 1 ( 0-100.0rpm Volts) ==========================================
//EA601 : trocado por momento pela saida: VEL_ALT1 
converteEA601(IN:=VEL_ALT1 , IN_MIN:=0000, IN_MAX:=100,OUT_MIN:=0, OUT_MAX:=1750);
LEITURA_VEL_ALT1:= converteEA601.OUT;


// Entrada analógica 7 : NX6000_1 - Leitura velocidade bomba alta 2 ( rpm Volts) =================================================
//EA701 : trocado por momento pela saida: VEL_ALT2
converteEA701(IN:=VEL_ALT2, IN_MIN:=0000, IN_MAX:=100,OUT_MIN:=0, OUT_MAX:=1750);
LEITURA_VEL_ALT2:= converteEA701.OUT;


// Entrada analógica 8 : NX6000_1 - Leitura presão da torre ( mma mA) ===================================================== 
converteEA801(IN:=EA801, IN_MIN:=0000, IN_MAX:=4000,OUT_MIN:=-125, OUT_MAX:=125);
LEITURA_PRES_TORRE:= converteEA801.OUT;


// Entrada analógica 1 : NX6000_2 - Leitura peso fluidizador 1 ( kg mA) ===================================================== 
converteEA102(IN:=EA102, IN_MIN:=799, IN_MAX:=4000,OUT_MIN:=0, OUT_MAX:=2000);
LEITURA_PESO_FLUI1_INST:= converteEA102.OUT;

//Filtro de amostragem peso do Fluidizador 1
BLINK_0(ENABLE:= TRUE, TIMELOW:= T#10S, TIMEHIGH:= T#5S, OUT=> HABIL_ATUAL_FLUI1);
IF HABIL_ATUAL_FLUI1 THEN
	LEITURA_PESO_FLUI1:= LEITURA_PESO_FLUI1_INST;
END_IF


// Entrada analógica 2 : NX6000_2 - Leitura peso fluidizador 2 ( kg mA) ===================================================== 
converteEA202(IN:=EA202, IN_MIN:=799, IN_MAX:=4000,OUT_MIN:=0, OUT_MAX:=2000);
LEITURA_PESO_FLUI2_INST:= converteEA202.OUT;
//Filtro de amostragem peso do Fluidizador 2
BLINK_1(ENABLE:= TRUE, TIMELOW:= T#10S, TIMEHIGH:= T#5S, OUT=> HABIL_ATUAL_FLUI2);
IF HABIL_ATUAL_FLUI2 THEN
	LEITURA_PESO_FLUI2:= LEITURA_PESO_FLUI2_INST;
END_IF
//======ROBY======ROBY=========ROBY=========ROBY=========ROBY======ROBY=========ROBY=========ROBY=======
// Entrada analógica 3 : NX6000_2 - Medição de umidade ======================================================= 
converteEA402(IN:=EA402, IN_MIN:=0, IN_MAX:=4000,OUT_MIN:=0, OUT_MAX:=13);
VALOR_MEDICAO_UMIDADE:= converteEA402.OUT;

// Entrada analógica 02 : NX6000_2 - %IW51 - Medição da temperatura da TORRE com PT100 e TXBLOCK =========================== 
converteEA303(IN:=EA303, IN_MIN:=0, IN_MAX:=4000,OUT_MIN:=0, OUT_MAX:=200);
TEMP_TORRE:= converteEA303.OUT;

